# B&R Automation Studio project CControl_Gschneitner (part 2)

### Parameter.typ
```iecst
TYPE
	parAnlage : {REDUND_UNREPLICABLE} 	STRUCT
		Allgemein : {REDUND_UNREPLICABLE} parAllgemein;
		Betrieb : {REDUND_UNREPLICABLE} parBetrieb;
		Ausstattung : {REDUND_UNREPLICABLE} parAusstattung;
		Schrittkette : {REDUND_UNREPLICABLE} parSchrittkette;
		Ventilator1 : {REDUND_UNREPLICABLE} parVentilator;
		Ventilator2 : {REDUND_UNREPLICABLE} parVentilator;
		Boxen : {REDUND_UNREPLICABLE} ARRAY[1..6]OF parBoxen;
		Entfeuchter : {REDUND_UNREPLICABLE} parEntfeuchter;
		Kompressor1 : {REDUND_UNREPLICABLE} parKompressor;
		Kompressor2 : {REDUND_UNREPLICABLE} parKompressor;
		Warmluftofen : {REDUND_UNREPLICABLE} parWarmluftofen;
		Heizregister : {REDUND_UNREPLICABLE} parHeizregister;
		Abluftventilator : {REDUND_UNREPLICABLE} parAbluftventilator;
		Abluftklappe : {REDUND_UNREPLICABLE} parAbluftklappe;
		Umschaltklappen : {REDUND_UNREPLICABLE} parUmschaltklappen;
		Bypassklappe : {REDUND_UNREPLICABLE} parBypassklappe;
		KlappenBoxen : {REDUND_UNREPLICABLE} ARRAY[1..6]OF parKlappenBoxen;
		Notstromaggregat : {REDUND_UNREPLICABLE} parNotstromaggregat;
		Sensoren : {REDUND_UNREPLICABLE} parSensoren;
		Servicebereich : {REDUND_UNREPLICABLE} parServicebereich;
		Fernalarmierung : {REDUND_UNREPLICABLE} parFernalarmierung;
		Scheitholzofen : {REDUND_UNREPLICABLE} parScheitholzofen;
		Tarifabschaltung : {REDUND_UNREPLICABLE} parTarifabschaltung;
		Strombegrenzung : {REDUND_UNREPLICABLE} parStrombegrenzung;
		SchlechtwetterBoxen : {REDUND_UNREPLICABLE} ARRAY[1..6]OF parSchlechtwetterBoxen;
	END_STRUCT;
	parAllgemein : {REDUND_UNREPLICABLE} 	STRUCT
		IPAdresse : {REDUND_UNREPLICABLE} STRING[16];
		SubnetMask : {REDUND_UNREPLICABLE} STRING[16];
		DefaultGateway : {REDUND_UNREPLICABLE} STRING[16];
		HostName : {REDUND_UNREPLICABLE} STRING[16];
		DatumUhrzeitLetzterBetrieb : {REDUND_UNREPLICABLE} DATE_AND_TIME;
		VerzoegerungWarnungen : {REDUND_UNREPLICABLE} REAL;
		VerzoegerungFehler : {REDUND_UNREPLICABLE} REAL;
		StandortHoehe : {REDUND_UNREPLICABLE} REAL;
		AnsaugflaecheVent : {REDUND_UNREPLICABLE} REAL; (*Ansaugfläche des Ventilators (für Luftmengenregelung ohne Entfeuchter)*)
		VerzoegerungAenderungKlappen : {REDUND_UNREPLICABLE} UDINT;
		LoginTimeout : {REDUND_UNREPLICABLE} UDINT;
		VerzUmschBetriebsartBoxen : {REDUND_UNREPLICABLE} UDINT;
		DisplayTimeout : {REDUND_UNREPLICABLE} INT;
		Sprache : {REDUND_UNREPLICABLE} USINT;
		PasswortschutzAus : {REDUND_UNREPLICABLE} BOOL;
		AutoLogoutEin : {REDUND_UNREPLICABLE} BOOL;
		ParameterVorhanden : {REDUND_UNREPLICABLE} BOOL; (*Wenn FALSE, wird beim Neustart der Standardparametersatz geladen*)
	END_STRUCT;
	parBetrieb : {REDUND_UNREPLICABLE} 	STRUCT
		BetriebAutoEin : {REDUND_UNREPLICABLE} BOOL;
	END_STRUCT;
	parAusstattung : {REDUND_UNREPLICABLE} 	STRUCT
		Ventilator1 : {REDUND_UNREPLICABLE} BOOL := TRUE;
		Ventilator2 : {REDUND_UNREPLICABLE} BOOL;
		Entfeuchter : {REDUND_UNREPLICABLE} BOOL;
		EntfeuchterFremd : {REDUND_UNREPLICABLE} BOOL;
		Warmluftofen : {REDUND_UNREPLICABLE} BOOL;
		WarmluftofenBetriebsmldg : {REDUND_UNREPLICABLE} BOOL;
		WarmluftofenTempVorgabe : {REDUND_UNREPLICABLE} BOOL;
		Heizregister : {REDUND_UNREPLICABLE} BOOL;
		HeizregisterDrehzahlvorgabe : {REDUND_UNREPLICABLE} BOOL;
		Scheitholzofen : {REDUND_UNREPLICABLE} BOOL;
		Notstromaggregat : {REDUND_UNREPLICABLE} BOOL;
		Energiemessung : {REDUND_UNREPLICABLE} BOOL;
		Bypassklappe : {REDUND_UNREPLICABLE} BOOL;
		Umschaltklappe1 : {REDUND_UNREPLICABLE} BOOL;
		Umschaltklappe2 : {REDUND_UNREPLICABLE} BOOL;
		Brandschutzklappe : {REDUND_UNREPLICABLE} BOOL;
		Abluftklappe : {REDUND_UNREPLICABLE} BOOL;
		Abluftventilator : {REDUND_UNREPLICABLE} BOOL;
		SensorFrischluft : {REDUND_UNREPLICABLE} BOOL;
		SensorDachluft : {REDUND_UNREPLICABLE} BOOL;
		SensorTrockenluft : {REDUND_UNREPLICABLE} BOOL;
		SensorAbluft : {REDUND_UNREPLICABLE} BOOL;
		SensorLuftgeschwindigkeit : {REDUND_UNREPLICABLE} BOOL;
		SensorKanaldruck : {REDUND_UNREPLICABLE} BOOL;
		Box1 : {REDUND_UNREPLICABLE} BOOL := TRUE;
		Box2 : {REDUND_UNREPLICABLE} BOOL;
		Box3 : {REDUND_UNREPLICABLE} BOOL;
		Box4 : {REDUND_UNREPLICABLE} BOOL;
		Box5 : {REDUND_UNREPLICABLE} BOOL;
		Box6 : {REDUND_UNREPLICABLE} BOOL;
		AlleBoxenklSchliessenWennAus : {REDUND_UNREPLICABLE} BOOL; (*Wenn aktiv, werden alle angesteuerten Boxenklappen im Stillstand geschlossen*)
		MehrereBoxenBelueftbar : {REDUND_UNREPLICABLE} BOOL;
		LuftmngReglerFrischlVent1 : {REDUND_UNREPLICABLE} BOOL; (*Auswahl, ob Luftmengenregelung im Frischluft/Dachluftbetrieb bei Ventilator 1 möglich*)
		LuftmngReglerUmluftVent1 : {REDUND_UNREPLICABLE} BOOL; (*Auswahl, ob Luftmengenregelung im Umluftbetrieb bei Ventilator 1 möglich*)
		LuftmngReglerFrischlVent2 : {REDUND_UNREPLICABLE} BOOL; (*Auswahl, ob Luftmengenregelung im Frischluft/Dachluftbetrieb bei Ventilator 2 möglich*)
		LuftmngReglerUmluftVent2 : {REDUND_UNREPLICABLE} BOOL; (*Auswahl, ob Luftmengenregelung im Umluftbetrieb bei Ventilator 2 möglich*)
		EntfeuchterNurImUmluftbetrieb : {REDUND_UNREPLICABLE} BOOL; (*Betrieb des Entfeuchters ist nur im Umluftbetrieb möglich*)
		BeideVentAusBeiUmschBypasskl : {REDUND_UNREPLICABLE} BOOL; (*Wenn TRUE, wird die Drehzahl beider Ventilatoren bei Umschaltung der Bypassklappe reduziert*)
		BeideVentAusBeiUmschBoxenkl : {REDUND_UNREPLICABLE} BOOL; (*Wenn TRUE, wird die Drehzahl beider Ventilatoren bei Umschaltung der Boxenklappen reduziert*)
		Vent1AusWennUmschUmluftkl : {REDUND_UNREPLICABLE} BOOL; (*Wenn TRUE, wird die Drehzahl von Ventilator 1 bei Umschaltung Umluftklappen reduziert*)
		Vent2AusWennUmschUmluftkl : {REDUND_UNREPLICABLE} BOOL; (*Wenn TRUE, wird die Drehzahl von Ventilator 2 bei Umschaltung Umluftklappen reduziert*)
		AbluftklImFrischlbetrImmerOffen : {REDUND_UNREPLICABLE} BOOL; (*Wenn TRUE, wird die Abluftklappe im Frischluftbetrieb immer geöffnet (im Automatikbetrieb der Klappe)*)
		StellungUmluftklappe1Stillstand : {REDUND_UNREPLICABLE} BOOL; (*FALSE= Frischluft, TRUE= Umluft*)
		StellungUmluftklappe2Stillstand : {REDUND_UNREPLICABLE} BOOL; (*FALSE= Frischluft, TRUE= Umluft*)
		EndlagenVhdUmschaltklappe1 : {REDUND_UNREPLICABLE} BOOL; (*Option Endlagen: Sind keine Endlagen vorhanden, wird die Klappe für die eingestellte Laufzeit umgeschaltet.*)
		EndlagenVhdUmschaltklappe2 : {REDUND_UNREPLICABLE} BOOL; (*Option Endlagen: Sind keine Endlagen vorhanden, wird die Klappe für die eingestellte Laufzeit umgeschaltet.*)
		EndlagenVhdBypassklappe : {REDUND_UNREPLICABLE} BOOL; (*Option Endlagen: Sind keine Endlagen vorhanden, wird die Klappe für die eingestellte Laufzeit umgeschaltet.*)
		EndlagenVhdBoxenklappe1 : {REDUND_UNREPLICABLE} BOOL; (*Option Endlagen: Sind keine Endlagen vorhanden, wird die Klappe für die eingestellte Laufzeit umgeschaltet.*)
		EndlagenVhdBoxenklappe2 : {REDUND_UNREPLICABLE} BOOL; (*Option Endlagen: Sind keine Endlagen vorhanden, wird die Klappe für die eingestellte Laufzeit umgeschaltet.*)
		EndlagenVhdBoxenklappe3 : {REDUND_UNREPLICABLE} BOOL; (*Option Endlagen: Sind keine Endlagen vorhanden, wird die Klappe für die eingestellte Laufzeit umgeschaltet.*)
		EndlagenVhdBoxenklappe4 : {REDUND_UNREPLICABLE} BOOL; (*Option Endlagen: Sind keine Endlagen vorhanden, wird die Klappe für die eingestellte Laufzeit umgeschaltet.*)
		EndlagenVhdBoxenklappe5 : {REDUND_UNREPLICABLE} BOOL; (*Option Endlagen: Sind keine Endlagen vorhanden, wird die Klappe für die eingestellte Laufzeit umgeschaltet.*)
		EndlagenVhdBoxenklappe6 : {REDUND_UNREPLICABLE} BOOL; (*Option Endlagen: Sind keine Endlagen vorhanden, wird die Klappe für die eingestellte Laufzeit umgeschaltet.*)
	END_STRUCT;
	parSchrittkette : {REDUND_UNREPLICABLE} 	STRUCT
		AnlaufverzZweiterVentilator : {REDUND_UNREPLICABLE} UDINT;
		VerzWetterwechsel : {REDUND_UNREPLICABLE} UDINT;
	END_STRUCT;
	parVentilator : {REDUND_UNREPLICABLE} 	STRUCT
		LuftmengeSollFrischluft : {REDUND_UNREPLICABLE} REAL; (*Soll-Luftmenge im Frischluftbetrieb in m³/h pro m² Boxenfläche*)
		LuftmengeSollUmluft : {REDUND_UNREPLICABLE} REAL; (*Soll-Luftmenge im Umluftbetrieb in m³/h pro m² Boxenfläche*)
		LuftmengeBoxMin : {REDUND_UNREPLICABLE} REAL; (*Minimale Lufmenge pro m² Boxenfläche in m³/h*)
		LuftmengeBoxMax : {REDUND_UNREPLICABLE} REAL; (*Maximale Lufmenge pro m² Boxenfläche in m³/h*)
		DrehzahlMin : {REDUND_UNREPLICABLE} REAL; (*Minimale Drehzahl des Ventilators [%]*)
		DrehzahlMax : {REDUND_UNREPLICABLE} REAL; (*Maximale Drehzahl des Ventilators [%]*)
		DrehzahlBeiAuskuehlphase : {REDUND_UNREPLICABLE} REAL; (*Soll-Drehzahl, wenn keine Box aktiv und WLO oder SHO noch in Betrieb [%]*)
		DrzUmschaltung : {REDUND_UNREPLICABLE} REAL; (*Soll-Drehzahl bei Klappenumschaltungen, wenn keine Luftaufbereitung in Betrieb ist [%]*)
		DrzUmschaltungMitLuftaufb : {REDUND_UNREPLICABLE} REAL; (*Soll-Drehzahl bei Klappenumschaltungen, wenn Luftaufbereitung in Betrieb ist [%]*)
		DrehzahlFixUmluft : {REDUND_UNREPLICABLE} REAL; (*Fix-Drehzahl bei Umluftbetrieb [%]*)
		DrehzahlFixFrischluft : {REDUND_UNREPLICABLE} REAL; (*Fix-Drehzahl bei Frischluftbetrieb [%]*)
		DrehzahlStrombegrenzung : {REDUND_UNREPLICABLE} REAL; (*Maximale Drehzahl, wenn Zeitfenster Strombegrenzung aktiv ist [%]*)
		DrehzahlLeistungsreduz : {REDUND_UNREPLICABLE} REAL; (*Maximale Drehzahl, wenn digitaler Eingang für Leistungsreduzierung aktiv ist [%]*)
		P : {REDUND_UNREPLICABLE} REAL;
		I : {REDUND_UNREPLICABLE} REAL;
		D : {REDUND_UNREPLICABLE} REAL;
		D_Filter : {REDUND_UNREPLICABLE} REAL;
		Hysterese : {REDUND_UNREPLICABLE} REAL;
		WindupDaempfung : {REDUND_UNREPLICABLE} REAL;
		Fehlerverzoegerung : {REDUND_UNREPLICABLE} REAL;
		ZeitRampeUp : {REDUND_UNREPLICABLE} UDINT; (*Rampenzeit UP [s]*)
		ZeitRampeDown : {REDUND_UNREPLICABLE} UDINT; (*Rampenzeit DOWN [s]*)
		LuftmengenregUmluftEin : {REDUND_UNREPLICABLE} BOOL; (*Wenn Ein, ist die Luftmengenregelung im Umluftbetrieb aktiv*)
		LuftmengenregFrischluftEin : {REDUND_UNREPLICABLE} BOOL; (*Wenn Ein, ist die Luftmengenregelung im Frischluftbetrieb aktiv*)
	END_STRUCT;
	parBoxen : {REDUND_UNREPLICABLE} 	STRUCT
		StellungKlappe1 : {REDUND_UNREPLICABLE} enumStellungKlappenBoxen; (*0= nicht verwendet, 1= geschlossen, 2= offen*)
		StellungKlappe2 : {REDUND_UNREPLICABLE} enumStellungKlappenBoxen; (*0= nicht verwendet, 1= geschlossen, 2= offen*)
		StellungKlappe3 : {REDUND_UNREPLICABLE} enumStellungKlappenBoxen; (*0= nicht verwendet, 1= geschlossen, 2= offen*)
		StellungKlappe4 : {REDUND_UNREPLICABLE} enumStellungKlappenBoxen; (*0= nicht verwendet, 1= geschlossen, 2= offen*)
		StellungKlappe5 : {REDUND_UNREPLICABLE} enumStellungKlappenBoxen; (*0= nicht verwendet, 1= geschlossen, 2= offen*)
		StellungKlappe6 : {REDUND_UNREPLICABLE} enumStellungKlappenBoxen; (*0= nicht verwendet, 1= geschlossen, 2= offen*)
		Grundflaeche : {REDUND_UNREPLICABLE} REAL; (*Grundfläche Box bei Losetrocknung in m²*)
		NameBox : {REDUND_UNREPLICABLE} STRING[20]; (*Name der Box*)
		Trockengut : {REDUND_UNREPLICABLE} USINT; (*0 = Heu (Lose), 1= Rundballen, 2= Mais, 3= Getreide, 4= Hopfen, 5= Kräuter, 6= Holz*)
		Aus : {REDUND_UNREPLICABLE} BOOL; (*Box Ausgeschaltet*)
		DauerbetriebEin : {REDUND_UNREPLICABLE} BOOL; (*Betriebsart Dauerbetrieb Ein*)
		IntervallbetriebEin : {REDUND_UNREPLICABLE} BOOL; (*Betriebsart Intervallbetrieb Ein*)
		NachtrocknungEin : {REDUND_UNREPLICABLE} BOOL; (*Betriebsart Nachtrocknung Ein*)
		Ventilator1 : {REDUND_UNREPLICABLE} BOOL; (*0= nicht für Box zuständig, 1= für Box zuständig*)
		Ventilator2 : {REDUND_UNREPLICABLE} BOOL; (*0= nicht für Box zuständig, 1= für Box zuständig*)
		Luftentfeuchter : {REDUND_UNREPLICABLE} BOOL; (*0= nicht für Box zuständig, 1= für Box zuständig*)
		Warmluftofen : {REDUND_UNREPLICABLE} BOOL; (*0= nicht für Box zuständig, 1= für Box zuständig*)
		Heizregister : {REDUND_UNREPLICABLE} BOOL; (*0= nicht für Box zuständig, 1= für Box zuständig*)
		Scheitholzofen : {REDUND_UNREPLICABLE} BOOL; (*0= nicht für Box zuständig, 1= für Box zuständig*)
		IntervallbetriebZeiten : {REDUND_UNREPLICABLE} ARRAY[0..23]OF BOOL; (*Zeitbereiche 0-23h Intervallbetrieb*)
		NachtrocknungZeiten : {REDUND_UNREPLICABLE} ARRAY[0..23]OF BOOL; (*Zeitbereiche 0-23h Nachtrocknungsbetrieb*)
	END_STRUCT;
	parZeitfenster : {REDUND_UNREPLICABLE} 	STRUCT
		StartStd : {REDUND_UNREPLICABLE} USINT;
		StartMin : {REDUND_UNREPLICABLE} USINT;
		StoppStd : {REDUND_UNREPLICABLE} USINT;
		StoppMin : {REDUND_UNREPLICABLE} USINT;
	END_STRUCT;
	parEntfeuchter : {REDUND_UNREPLICABLE} 	STRUCT
		Type : {REDUND_UNREPLICABLE} ARRAY[0..14]OF STRING[20];
		Registerflaeche : {REDUND_UNREPLICABLE} ARRAY[0..14]OF REAL;
		EinschaltverzKompressor : {REDUND_UNREPLICABLE} UDINT;
		EinschaltverzAbtau : {REDUND_UNREPLICABLE} UDINT;
		MindestlaufzeitOelsumpf : {REDUND_UNREPLICABLE} UDINT;
		MaxZeitStromlos : {REDUND_UNREPLICABLE} UDINT;
		RestzeitLaufzOelsumpf : {REDUND_UNREPLICABLE} UDINT;
		AnlaufverzModul2 : {REDUND_UNREPLICABLE} UDINT;
		AusschaltverzAbtau : {REDUND_UNREPLICABLE} UDINT;
		LuftgeschwEntfeuchterMin : {REDUND_UNREPLICABLE} REAL; (*Minimale Luftgeschwindigkeit über den Entfeuchter in m/s*)
		LuftgeschwEntfeuchterMax : {REDUND_UNREPLICABLE} REAL; (*Maximale Luftgeschwindigkeit über den Entfeuchter in m/s*)
		EintrittFeuchteEin : {REDUND_UNREPLICABLE} REAL;
		EintrittFeuchteAus : {REDUND_UNREPLICABLE} REAL;
		Dauerbetrieb : {REDUND_UNREPLICABLE} BOOL;
		Automatikbetrieb : {REDUND_UNREPLICABLE} BOOL;
		Aus : {REDUND_UNREPLICABLE} BOOL;
		IndexType : {REDUND_UNREPLICABLE} USINT;
		VerzStandbyHochdruckMax : {REDUND_UNREPLICABLE} UDINT; (*Wenn während Klappenumschaltung oder Strombegrenzung Ventilator Hochdruck überschritten -> Standby*)
		VerzBetriebsmeldung : {REDUND_UNREPLICABLE} UDINT; (*Nur für Fremdgeräte in Verwendung*)
	END_STRUCT;
	parKompressor : {REDUND_UNREPLICABLE} 	STRUCT
		EinschaltverzMagnetventil : {REDUND_UNREPLICABLE} UDINT;
		DrehzahlMin : {REDUND_UNREPLICABLE} REAL;
		DrehzahlMax : {REDUND_UNREPLICABLE} REAL;
		NiederdruckMin : {REDUND_UNREPLICABLE} REAL;
		NiederdruckMax : {REDUND_UNREPLICABLE} REAL;
		RampeDown : {REDUND_UNREPLICABLE} REAL;
		RampeUp : {REDUND_UNREPLICABLE} REAL;
		NiederdruckPumpDown : {REDUND_UNREPLICABLE} REAL;
		DrehzahlFix : {REDUND_UNREPLICABLE} REAL;
		DrehzahlReduzierung : {REDUND_UNREPLICABLE} REAL;
		EintrittTempMin : {REDUND_UNREPLICABLE} REAL;
		EintrittTempMax : {REDUND_UNREPLICABLE} REAL;
		HochdruckMax : {REDUND_UNREPLICABLE} REAL;
		NiederdruckSoll : {REDUND_UNREPLICABLE} REAL;
		Hysterese : {REDUND_UNREPLICABLE} REAL;
		P : {REDUND_UNREPLICABLE} REAL;
		I : {REDUND_UNREPLICABLE} REAL;
		D : {REDUND_UNREPLICABLE} REAL;
		DrehzahlregelungEin : {REDUND_UNREPLICABLE} BOOL;
	END_STRUCT;
	parWarmluftofen : {REDUND_UNREPLICABLE} 	STRUCT
		SaettigungFrischlEin : {REDUND_UNREPLICABLE} REAL;
		WarmlufttempVorgabeSoll : {REDUND_UNREPLICABLE} REAL;
		Hysterese : {REDUND_UNREPLICABLE} REAL;
		Auskuehlzeit : {REDUND_UNREPLICABLE} UDINT;
		VerzBetriebsmeldung : {REDUND_UNREPLICABLE} UDINT;
		VerzWetterwechsel : {REDUND_UNREPLICABLE} UDINT;
		DauerbetriebEin : {REDUND_UNREPLICABLE} BOOL;
		AutomatikbetriebEin : {REDUND_UNREPLICABLE} BOOL;
		Aus : {REDUND_UNREPLICABLE} BOOL;
	END_STRUCT;
	parHeizregister : {REDUND_UNREPLICABLE} 	STRUCT
		VerzWetterwechsel : {REDUND_UNREPLICABLE} UDINT;
		SaettigungFrischlEin : {REDUND_UNREPLICABLE} REAL;
		TrockenluftTempSoll : {REDUND_UNREPLICABLE} REAL;
		Hysterese : {REDUND_UNREPLICABLE} REAL;
		DrehzahlVorgabeMin : {REDUND_UNREPLICABLE} REAL;
		DrehzahlVorgabeMax : {REDUND_UNREPLICABLE} REAL;
		P : {REDUND_UNREPLICABLE} REAL;
		I : {REDUND_UNREPLICABLE} REAL;
		D : {REDUND_UNREPLICABLE} REAL;
		Aus : {REDUND_UNREPLICABLE} BOOL;
		DauerbetriebEin : {REDUND_UNREPLICABLE} BOOL;
		AutomatikbetriebEin : {REDUND_UNREPLICABLE} BOOL;
	END_STRUCT;
	parAbluftventilator : {REDUND_UNREPLICABLE} 	STRUCT
		AbluftfeuchteMax : {REDUND_UNREPLICABLE} REAL;
		Hysterese : {REDUND_UNREPLICABLE} REAL;
		DrehzahlMin : {REDUND_UNREPLICABLE} REAL;
		DrehzahlMax : {REDUND_UNREPLICABLE} REAL;
		P : {REDUND_UNREPLICABLE} REAL;
		I : {REDUND_UNREPLICABLE} REAL;
		D : {REDUND_UNREPLICABLE} REAL;
		Ein : {REDUND_UNREPLICABLE} BOOL;
		Automatik : {REDUND_UNREPLICABLE} BOOL;
	END_STRUCT;
	parAbluftklappe : {REDUND_UNREPLICABLE} 	STRUCT
		Laufzeit : {REDUND_UNREPLICABLE} UDINT;
		AbluftfeuchteMax : {REDUND_UNREPLICABLE} REAL;
		Hysterese : {REDUND_UNREPLICABLE} REAL;
		Automatik : {REDUND_UNREPLICABLE} BOOL;
		Oeffnen : {REDUND_UNREPLICABLE} BOOL;
		Schliessen : {REDUND_UNREPLICABLE} BOOL;
	END_STRUCT;
	parUmschaltklappen : {REDUND_UNREPLICABLE} 	STRUCT
		LaufzeitKlappe1 : {REDUND_UNREPLICABLE} UDINT;
		LaufzeitKlappe2 : {REDUND_UNREPLICABLE} UDINT;
		TemperaturUmschaltung : {REDUND_UNREPLICABLE} REAL;
		Hysterese : {REDUND_UNREPLICABLE} REAL;
		Umschaltverzoegerung : {REDUND_UNREPLICABLE} UDINT;
		TempDifferenzUmschaltung : {REDUND_UNREPLICABLE} REAL;
		Automatik : {REDUND_UNREPLICABLE} BOOL;
		Umluft : {REDUND_UNREPLICABLE} BOOL;
		Frischluft : {REDUND_UNREPLICABLE} BOOL;
	END_STRUCT;
	parBypassklappe : {REDUND_UNREPLICABLE} 	STRUCT
		Laufzeit : {REDUND_UNREPLICABLE} UDINT;
		Automatik : {REDUND_UNREPLICABLE} BOOL;
		Oeffnen : {REDUND_UNREPLICABLE} BOOL;
		Schliessen : {REDUND_UNREPLICABLE} BOOL;
	END_STRUCT;
	parKlappenBoxen : {REDUND_UNREPLICABLE} 	STRUCT
		Laufzeit : {REDUND_UNREPLICABLE} UDINT;
	END_STRUCT;
	parNotstromaggregat : {REDUND_UNREPLICABLE} 	STRUCT
		Vorlaufzeit : {REDUND_UNREPLICABLE} UDINT;
		VerzBetriebsmeldung : {REDUND_UNREPLICABLE} UDINT;
		Nachlaufzeit : {REDUND_UNREPLICABLE} UDINT;
	END_STRUCT;
	parSensoren : {REDUND_UNREPLICABLE} 	STRUCT
		NiederdruckMessberMin : {REDUND_UNREPLICABLE} REAL;
		NiederdruckMessberMax : {REDUND_UNREPLICABLE} REAL;
		HochdruckMessberMin : {REDUND_UNREPLICABLE} REAL;
		HochdruckMessberMax : {REDUND_UNREPLICABLE} REAL;
		EintrittTempMessberMin : {REDUND_UNREPLICABLE} REAL;
		EintrittTempMessberMax : {REDUND_UNREPLICABLE} REAL;
		EintrittFeuchteMessberMin : {REDUND_UNREPLICABLE} REAL;
		EintrittFeuchteMessberMax : {REDUND_UNREPLICABLE} REAL;
		AustrittTempMessberMin : {REDUND_UNREPLICABLE} REAL;
		AustrittTempMessberMax : {REDUND_UNREPLICABLE} REAL;
		AustrittFeuchteMessberMin : {REDUND_UNREPLICABLE} REAL;
		AustrittFeuchteMessberMax : {REDUND_UNREPLICABLE} REAL;
		FrischlTempMessberMin : {REDUND_UNREPLICABLE} REAL;
		FrischlTempMessberMax : {REDUND_UNREPLICABLE} REAL;
		FrischlFeuchteMessberMin : {REDUND_UNREPLICABLE} REAL;
		FrischlFeuchteMessberMax : {REDUND_UNREPLICABLE} REAL;
		DachTempMessberMin : {REDUND_UNREPLICABLE} REAL;
		DachTempMessberMax : {REDUND_UNREPLICABLE} REAL;
		DachFeuchteMessberMin : {REDUND_UNREPLICABLE} REAL;
		DachFeuchteMessberMax : {REDUND_UNREPLICABLE} REAL;
		TrockenlTempMessberMin : {REDUND_UNREPLICABLE} REAL;
		TrockenlTempMessberMax : {REDUND_UNREPLICABLE} REAL;
		TrockenlFeuchteMessberMin : {REDUND_UNREPLICABLE} REAL;
		TrockenlFeuchteMessberMax : {REDUND_UNREPLICABLE} REAL;
		AbluftTempMessberMin : {REDUND_UNREPLICABLE} REAL;
		AbluftTempMessberMax : {REDUND_UNREPLICABLE} REAL;
		AbluftFeuchteMessberMin : {REDUND_UNREPLICABLE} REAL;
		AbluftFeuchteMessberMax : {REDUND_UNREPLICABLE} REAL;
		KanaldruckMessberMin : {REDUND_UNREPLICABLE} REAL;
		KanaldruckMessberMax : {REDUND_UNREPLICABLE} REAL;
		LuftgeschwMessberMin : {REDUND_UNREPLICABLE} REAL;
		LuftgeschwMessberMax : {REDUND_UNREPLICABLE} REAL;
		OffsetNiederdruckModul1 : {REDUND_UNREPLICABLE} REAL;
		OffsetNiederdruckModul2 : {REDUND_UNREPLICABLE} REAL;
		OffsetHochdruckModul1 : {REDUND_UNREPLICABLE} REAL;
		OffsetHochdruckModul2 : {REDUND_UNREPLICABLE} REAL;
		OffsetEintrittTemp : {REDUND_UNREPLICABLE} REAL;
		OffsetEintrittFeuchte : {REDUND_UNREPLICABLE} REAL;
		OffsetAustrittTemp : {REDUND_UNREPLICABLE} REAL;
		OffsetAustrittFeuchte : {REDUND_UNREPLICABLE} REAL;
		OffsetFrischluftTemp : {REDUND_UNREPLICABLE} REAL;
		OffsetFrischluftFeuchte : {REDUND_UNREPLICABLE} REAL;
		OffsetDachTemp : {REDUND_UNREPLICABLE} REAL;
		OffsetDachFeuchte : {REDUND_UNREPLICABLE} REAL;
		OffsetTrockenluftTemp : {REDUND_UNREPLICABLE} REAL;
		OffsetTrockenluftFeuchte : {REDUND_UNREPLICABLE} REAL;
		OffsetAbluftTemp : {REDUND_UNREPLICABLE} REAL;
		OffsetAbluftFeuchte : {REDUND_UNREPLICABLE} REAL;
		OffsetKanaldruck : {REDUND_UNREPLICABLE} REAL;
		OffsetLuftgeschw : {REDUND_UNREPLICABLE} REAL;
		FilterzeitNiederdruck : {REDUND_UNREPLICABLE} UINT;
		FilterzeitHochdruck : {REDUND_UNREPLICABLE} UINT;
		FilterzeitEintritt : {REDUND_UNREPLICABLE} UINT;
		FilterzeitAustritt : {REDUND_UNREPLICABLE} UINT;
		FilterzeitFrischluft : {REDUND_UNREPLICABLE} UINT;
		FilterzeitDachluft : {REDUND_UNREPLICABLE} UINT;
		FilterzeitTrockenluft : {REDUND_UNREPLICABLE} UINT;
		FilterzeitAbluft : {REDUND_UNREPLICABLE} UINT;
		FilterzeitKanaldruck : {REDUND_UNREPLICABLE} UINT;
		FilterzeitLuftgeschwindigkeit : {REDUND_UNREPLICABLE} UINT;
	END_STRUCT;
	parServicebereich : {REDUND_UNREPLICABLE} 	STRUCT
		KontrollintervallUhrzeit : {REDUND_UNREPLICABLE} UDINT;
	END_STRUCT;
	parFernalarmierung : {REDUND_UNREPLICABLE} 	STRUCT
		MailAdresse : {REDUND_UNREPLICABLE} ARRAY[0..3]OF STRING[80];
		EMailAlarmierungEin : {REDUND_UNREPLICABLE} BOOL;
	END_STRUCT;
	parScheitholzofen : {REDUND_UNREPLICABLE} 	STRUCT
		Auskuehlzeit : {REDUND_UNREPLICABLE} UDINT;
	END_STRUCT;
	parTarifabschaltung : {REDUND_UNREPLICABLE} 	STRUCT
		Zeitfenster : {REDUND_UNREPLICABLE} parZeitfenster;
		VorlaufzeitAbschaltungLuftaufb : {REDUND_UNREPLICABLE} USINT;
	END_STRUCT;
	parStrombegrenzung : {REDUND_UNREPLICABLE} 	STRUCT
		Zeitfenster : {REDUND_UNREPLICABLE} parZeitfenster;
	END_STRUCT;
	parSchlechtwetterBoxen : {REDUND_UNREPLICABLE} 	STRUCT
		Stufe : {REDUND_UNREPLICABLE} ARRAY[1..6]OF parSchlechtwetterBoxenStufen;
		HystereseGrenzwert : {REDUND_UNREPLICABLE} REAL;
		AuswahlSensorGrenzwert : {REDUND_UNREPLICABLE} USINT; (*Option Auswahl zuständiger Sensor für Grenzwert (0= Frischluft, 1= Dachluft, 2= Trockenluft)*)
		MaterialfeuchteIst : {REDUND_UNREPLICABLE} USINT; (*Aktuell Materialfeuchte (Trockengutfeuchte) der Box (%)*)
	END_STRUCT;
	parSchlechtwetterBoxenStufen : {REDUND_UNREPLICABLE} 	STRUCT
		Saettigungsdefizit : {REDUND_UNREPLICABLE} REAL; (*Grenzwert Sättigungsdefizit Schlechtwetter [g/m³]*)
		SchlechtwetterZeitLauf : {REDUND_UNREPLICABLE} UDINT; (*Laufzeit bei Schlechtwetter [ms]*)
		SchlechtwetterZeitPause : {REDUND_UNREPLICABLE} UDINT; (*Pausenzeit bei Schlechtwetter [ms]*)
		MaterialfeuchteStufe : {REDUND_UNREPLICABLE} UINT; (*Max. Trockengutfeuchte der Stufe (%)*)
	END_STRUCT;
END_TYPE
```

### Enumeration.typ
```iecst
TYPE
	enumStatusmeldungen :
		(
		STATUSMLDG_STILLSTAND := 0,
		STATUSMLDG_TESTBETRIEB := 1,
		STATUSMLDG_AUTOMATIKBETRIEB := 2,
		STATUSMLDG_DAUERBETRIEB := 3,
		STATUSMLDG_VENTILATOR_EIN := 4,
		STATUSMLDG_VENTILATOR_INTERV := 5
		);
	enumStatus :
		(
		STATUS_NICHT_VERFUEGBAR := 0,
		STATUS_STILLSTAND := 1,
		STATUS_TESTBETRIEB := 2,
		STATUS_DAUERBETRIEB := 3,
		STATUS_INTERVALL_LAUF := 4,
		STATUS_INTERVALL_PAUSE := 5,
		STATUS_NACHTROCKNUNG_LAUF := 6,
		STATUS_NACHTROCKNUNG_PAUSE := 7,
		STATUS_BEREIT := 8,
		STATUS_STOERUNG := 9,
		STATUS_AKTIV := 10,
		STATUS_NICHT_AKTIV := 11,
		STATUS_OFFEN := 12,
		STATUS_GESCHLOSSEN := 13,
		STATUS_NICHT_FREIGEGEBEN := 14,
		STATUS_UNBEKANNT := 15,
		STATUS_IN_BEWEGUNG := 16,
		STATUS_ENTF_ABTAUUNG := 17,
		STATUS_ANLAGE_IN_BETRIEB := 18,
		STATUS_AUSKUEHLPHASE := 19,
		STATUS_ENTF_STANDBY := 20,
		STATUS_KLAPPE_FRISCHLUFT := 21,
		STATUS_KLAPPE_DACHLUFT := 22,
		STATUS_KLAPPE_UMLUFT := 23,
		STATUS_DAUERBETRIEB_PAUSIERT := 24,
		STATUS_SCHLECHTWETTER_LAUF := 25,
		STATUS_SCHLECHTWETTER_PAUSE := 26
		);
	enumBetriebsmodus :
		(
		STILLSTAND := 0,
		BETRIEB := 1,
		IOTEST := 2
		);
	enumWarnung :
		(
		WARNUNG_HOCHDRUCK_MAX_MOD1 := 0,
		WARNUNG_HOCHDRUCK_MAX_MOD2 := 1,
		WARNUNG_SENSOR_AUSTRITT := 2,
		WARNUNG_HEIZREGISTER_FROSTSCHUTZ := 3
		);
	enumFehler :
		(
		FEHLER_24VDC := 0,
		FEHLER_FU_KOMPRESSOR_MODUL1 := 1,
		FEHLER_FU_KOMPRESSOR_MODUL2 := 2,
		FEHLER_BETRIEBSMLDG_KOMPR_MOD1 := 3,
		FEHLER_BETRIEBSMLDG_KOMPR_MOD2 := 4,
		FEHLER_BETRIEBSMLDG_VENTILATOR1 := 5,
		FEHLER_BETRIEBSMLDG_VENTILATOR2 := 6,
		FEHLER_BETRIEBSMLDG_ABLUFTVENT := 7,
		FEHLER_HOCHDRUCK_MODUL1 := 8,
		FEHLER_HOCHDRUCK_MODUL2 := 9,
		FEHLER_NIEDERDRUCK_MODUL1 := 10,
		FEHLER_NIEDERDRUCK_MODUL2 := 11,
		FEHLER_OELDRUCK_KOMPR_MOD1 := 12,
		FEHLER_OELDRUCK_KOMPR_MOD2 := 13,
		FEHLER_KOPFTEMP_KOMPR_MOD1 := 14,
		FEHLER_KOPFTEMP_KOMPR_MOD2 := 15,
		FEHLER_VOLLSCHUTZ_KOMPR_MOD1 := 16,
		FEHLER_VOLLSCHUTZ_KOMPR_MOD2 := 17,
		FEHLER_BETRIEBSMLDG_WARMLUFTOFEN := 18,
		FEHLER_BETRIEBSMLDG_NOTSTROM := 19,
		FEHLER_SENSOR_FRISCHLUFT := 20,
		FEHLER_SENSOR_DACHLUFT := 21,
		FEHLER_SENSOR_TROCKENLUFT := 22,
		FEHLER_SENSOR_ABLUFT := 23,
		FEHLER_SENSOR_EINTRITT := 24,
		FEHLER_SENSOR_AUSTRITT := 25,
		FEHLER_SENSOR_LUFTGESCHW := 26,
		FEHLER_SENSOR_KANALDRUCK := 27,
		FEHLER_SENSOR_NIEDERDRUCK_MOD1 := 28,
		FEHLER_SENSOR_NIEDERDRUCK_MOD2 := 29,
		FEHLER_SENSOR_HOCHDRUCK_MOD1 := 30,
		FEHLER_SENSOR_HOCHDRUCK_MOD2 := 31,
		FEHLER_ENDLAGEN_BYPASSKLAPPE := 32,
		FEHLER_ENDLAGEN_UMSCHALTKLAPPE1 := 33,
		FEHLER_ENDLAGEN_UMSCHALTKLAPPE2 := 34,
		FEHLER_ENDLAGEN_BOXENKLAPPE_1 := 35,
		FEHLER_ENDLAGEN_BOXENKLAPPE_2 := 36,
		FEHLER_ENDLAGEN_BOXENKLAPPE_3 := 37,
		FEHLER_ENDLAGEN_BOXENKLAPPE_4 := 38,
		FEHLER_ENDLAGEN_BOXENKLAPPE_5 := 39,
		FEHLER_ENDLAGEN_BOXENKLAPPE_6 := 40,
		FEHLER_ENDLAGEN_ABLUFTKLAPPE := 41,
		FEHLER_EINTRITT_TEMP_ZU_HOCH := 42,
		FEHLER_EINTRITT_TEMP_ZU_NIEDRIG := 43,
		FEHLER_LZ_PUMPDOWN_MOD1 := 44,
		FEHLER_LZ_PUMPDOWN_MOD2 := 45,
		FEHLER_DREHFELD := 46,
		FEHLER_ENTF_FREMD_STOERMELDUNG := 47,
		FEHLER_ENTF_FREMD_BETRMLDG := 48
		);
	enumAktor :
		(
		AKTOR_SCHRITTKETTE := 0,
		AKTOR_OELSUMPFHEIZUNG_MOD1 := 1,
		AKTOR_OELSUMPFHEIZUNG_MOD2 := 2,
		AKTOR_KOMPRESSOR_MOD1 := 3,
		AKTOR_KOMPRESSOR_MOD2 := 4,
		AKTOR_VENTILATOR_1 := 5,
		AKTOR_VENTILATOR_2 := 6,
		AKTOR_BYPASSKLAPPE := 7,
		AKTOR_UMSCHALTKLAPPE_1 := 8,
		AKTOR_UMSCHALTKLAPPE_2 := 9,
		AKTOR_MAGNETVENTIL_MOD1 := 10,
		AKTOR_MAGNETVENTIL_MOD2 := 11,
		AKTOR_KLAPPE_BOX_1 := 12,
		AKTOR_KLAPPE_BOX_2 := 13,
		AKTOR_KLAPPE_BOX_3 := 14,
		AKTOR_KLAPPE_BOX_4 := 15,
		AKTOR_KLAPPE_BOX_5 := 16,
		AKTOR_KLAPPE_BOX_6 := 17,
		AKTOR_ABLUFTKLAPPE := 18,
		AKTOR_ABLUFTVENTILATOR := 19,
		AKTOR_WARMLUFTOFEN := 20,
		AKTOR_HEIZREGISTER := 21,
		AKTOR_SCHEITHOLZOFEN := 22,
		AKTOR_NOTSTROMAGGREGAT := 23,
		AKTOR_BRANDSCHUTZKLAPPE := 24,
		AKTOR_ENTFEUCHTER_FREMD := 25
		);
	enumSystem :
		(
		FEHLER_IO_TEST_NICHT_FERTIG := 0,
		FEHLER_KOMMUNIKATION_DISPLAY_IO := 1
		);
	enumIcon :
		(
		ICON_VISIBLE := 0,
		ICON_HIDDEN := 1,
		ICON_GRAU := 2,
		ICON_GELB := 3,
		ICON_ROT := 4,
		TEXT_HELLGRAU := 5,
		TEXT_DUNKELGRAU := 6,
		TEXT_GELB := 7,
		TROCKENGUT_HEU_GRAU := 8,
		TROCKENGUT_HEU_GELB := 9,
		TROCKENGUT_RUNDB_GRAU := 10,
		TROCKENGUT_RUNDB_GELB := 11,
		TROCKENGUT_MAIS_GRAU := 12,
		TROCKENGUT_MAIS_GELB := 13,
		TROCKENGUT_GETREIDE_GRAU := 14,
		TROCKENGUT_GETREIDE_GELB := 15,
		TROCKENGUT_HOPFEN_GRAU := 16,
		TROCKENGUT_HOPFEN_GELB := 17,
		TROCKENGUT_KRAEUTER_GRAU := 18,
		TROCKENGUT_KRAEUTER_GELB := 19,
		TROCKENGUT_HOLZ_GRAU := 20,
		TROCKENGUT_HOLZ_GELB := 21,
		TASTE_ENTF_INSELBETR_GESPERRT := 22,
		TASTE_ENTF_INSELBETR_AUS := 23,
		TASTE_ENTF_INSELBETR_EIN := 24
		);
	enumPasswoerter :
		(
		PASSWORT_SPERRE := 0,
		PASSWORT_KUNDE := 4321,
		PASSWORT_LASCO := 21666,
		PASSWORT_ADMIN := 110588,
		PASSWORT_TAN_01 := 222508,
		PASSWORT_TAN_02 := 988036,
		PASSWORT_TAN_03 := 617545,
		PASSWORT_TAN_04 := 548124,
		PASSWORT_TAN_05 := 321642,
		PASSWORT_TAN_06 := 482409,
		PASSWORT_TAN_07 := 679341,
		PASSWORT_TAN_08 := 455576,
		PASSWORT_TAN_09 := 825468,
		PASSWORT_TAN_10 := 959563,
		PASSWORT_TAN_11 := 107316,
		PASSWORT_TAN_12 := 724578,
		PASSWORT_TAN_13 := 804211,
		PASSWORT_TAN_14 := 147228,
		PASSWORT_TAN_15 := 564299,
		PASSWORT_TAN_16 := 832285,
		PASSWORT_TAN_17 := 981185,
		PASSWORT_TAN_18 := 598284,
		PASSWORT_TAN_19 := 730460,
		PASSWORT_TAN_20 := 971962,
		PASSWORT_TAN_21 := 728589,
		PASSWORT_TAN_22 := 396271,
		PASSWORT_TAN_23 := 496146,
		PASSWORT_TAN_24 := 727556,
		PASSWORT_TAN_25 := 110312,
		PASSWORT_TAN_26 := 849433,
		PASSWORT_TAN_27 := 388439,
		PASSWORT_TAN_28 := 907081,
		PASSWORT_TAN_29 := 347765,
		PASSWORT_TAN_30 := 189196,
		PASSWORT_TAN_31 := 129436,
		PASSWORT_TAN_32 := 678825,
		PASSWORT_TAN_33 := 603382,
		PASSWORT_TAN_34 := 752548,
		PASSWORT_TAN_35 := 466127,
		PASSWORT_TAN_36 := 419810,
		PASSWORT_TAN_37 := 628991,
		PASSWORT_TAN_38 := 349832,
		PASSWORT_TAN_39 := 219361,
		PASSWORT_TAN_40 := 257082,
		PASSWORT_TAN_41 := 166753,
		PASSWORT_TAN_42 := 346634,
		PASSWORT_TAN_43 := 635178,
		PASSWORT_TAN_44 := 740794,
		PASSWORT_TAN_45 := 924143,
		PASSWORT_TAN_46 := 162952,
		PASSWORT_TAN_47 := 218710,
		PASSWORT_TAN_48 := 839073,
		PASSWORT_TAN_49 := 423623,
		PASSWORT_TAN_50 := 232733,
		PASSWORT_ZU_GROSS := 999999,
		PASSWORT_ADMIN_1 := 081190,
		PASSWORT_SERVICE := 8613,
		PASSWORT_KUNDE_1 := 1234
		);
	enumPasswortebenen :
		(
		EBENE_SPERRE := 0,
		EBENE_KUNDE := 1,
		EBENE_SERVICE := 2,
		EBENE_LASCO := 3,
		EBENE_ADMIN := 4
		);
	enumSeitenVisu :
		(
		_000_INIT := 0,
		_001_LOGIN := 1,
		_010_HM_UEBERSICHT := 10,
		_100_AL := 100,
		_101_AL := 101,
		_400_IW := 400,
		_401_IW := 401,
		_402_IW := 402,
		_403_IW := 403,
		_404_IW := 404,
		_600_SYS := 600,
		_610_SYS := 610,
		_620_SYS := 620,
		_630_SYS := 630,
		_631_SYS := 631,
		_632_SYS := 632,
		_640_SYS := 640,
		_641_SYS := 641,
		_650_SYS := 650,
		_660_SYS := 660,
		_670_SYS := 670,
		_700_SYS := 700,
		_710_SYS := 710,
		_711_SYS := 711,
		_712_SYS := 712,
		_713_SYS := 713,
		_714_SYS := 714,
		_715_SYS := 715,
		_716_SYS := 716,
		_717_SYS := 717,
		_720_SYS := 720,
		_721_SYS := 721,
		_722_SYS := 722,
		_723_SYS := 723,
		_724_SYS := 724,
		_730_SYS := 730,
		_731_SYS := 731,
		_732_SYS := 732,
		_740_SYS := 740,
		_741_SYS := 741,
		_742_SYS := 742,
		_750_SYS := 750,
		_751_SYS := 751,
		_752_SYS := 752,
		_760_SYS := 760,
		_770_SYS := 770,
		_780_SYS := 780,
		_781_SYS := 781,
		_782_SYS := 782,
		_783_SYS := 783,
		_790_SYS := 790,
		_800_TEST := 800,
		_810_TEST := 810,
		_811_TEST := 811,
		_812_TEST := 812,
		_820_TEST := 820,
		_821_TEST := 821,
		_822_TEST := 822,
		_823_TEST := 823,
		_824_TEST := 824,
		_825_TEST := 825,
		_830_TEST := 830,
		_831_TEST := 831,
		_832_TEST := 832,
		_840_TEST := 840,
		_841_TEST := 841,
		_842_TEST := 842,
		_850_TEST := 850,
		_851_TEST := 851,
		_852_TEST := 852,
		_860_TEST := 860,
		_861_TEST := 861
		);
	enumZusatzmeldungen :
		(
		ZM_STILLSTAND_IOTEST_NICHT_ABGE := 0,
		ZM_STILLSTAND_FEHLER := 1,
		ZM_STILLSTAND_BEREIT := 2,
		ZM_STILLSTAND_ENTF_NOCH_IN_BETR := 3,
		ZM_WARTE_AUF_NOTSTROM := 4,
		ZM_AUSKUEHLZEIT_WLO_AKTIV := 5,
		ZM_AUSKUEHLZEIT_SHO_AKTIV := 6,
		ZM_ANLAUFVERZ_VENT2_AKTIV := 7,
		ZM_ANLAUFVERZ_VENT1_AKTIV := 8,
		ZM_TARIFABSCHALTUNG_AKTIV := 9,
		ZM_STROMBEGRENZUNG_AKTIV := 10,
		ZM_KLAPPEN_WERDEN_UMGESCHALTET := 11,
		ZM_FRISCHLUFTBETRIEB := 12,
		ZM_DACHABSAUGUNGSBETRIEB := 13,
		ZM_UMLUFTBETRIEB := 14,
		ZM_WARTE_AUF_ANFORDERUNG_BOX := 15,
		ZM_STILLSTAND_FEHLERSTOPP := 16,
		ZM_FRISCHLUFTB_VLZ_TARIF := 17,
		ZM_DACHABSAUGUNGSB_VLZ_TARIF := 18,
		ZM_UMLUFTBETR_VLZ_TARIF := 19,
		ZM_INSELBETRIEB_AUS := 20,
		ZM_INSELBETRIEB_STANDBY := 21,
		ZM_INSELBETRIEB_AKTIV := 22,
		ZM_INSELBETRIEB_VENT_NICHT_AKTIV := 23
		);
END_TYPE
```

### VisuIO.typ - Local data types
```iecst
TYPE
	typHmiStatus : {REDUND_UNREPLICABLE} 	STRUCT
		CurUserLevel : {REDUND_UNREPLICABLE} enumPasswortebenen;
		CurPage : {REDUND_UNREPLICABLE} enumSeitenVisu;
		hmiPasswort : {REDUND_UNREPLICABLE} enumPasswoerter;
		Box1 : {REDUND_UNREPLICABLE} typHmiStatusBoxen;
		Box2 : {REDUND_UNREPLICABLE} typHmiStatusBoxen;
		Box3 : {REDUND_UNREPLICABLE} typHmiStatusBoxen;
		Box4 : {REDUND_UNREPLICABLE} typHmiStatusBoxen;
		Box5 : {REDUND_UNREPLICABLE} typHmiStatusBoxen;
		Box6 : {REDUND_UNREPLICABLE} typHmiStatusBoxen;
		Ventilator1 : {REDUND_UNREPLICABLE} typHmiStatusVentilator;
		Ventilator2 : {REDUND_UNREPLICABLE} typHmiStatusVentilator;
		Entfeuchter : {REDUND_UNREPLICABLE} typHmiStatusEntfeuchter;
		WarmluftScheitholzofen : {REDUND_UNREPLICABLE} typHmiStatusWarmluftScheitholz;
		Heizregister : {REDUND_UNREPLICABLE} typHmiStatusHeizregister;
		Brandschutzklappe : {REDUND_UNREPLICABLE} typHmiStatusBrandschutzklappe;
		Umluftklappen : {REDUND_UNREPLICABLE} typHmiStatusUmluftklappen;
		Bypassklappe : {REDUND_UNREPLICABLE} typHmiStatusBypassklappe;
		Abluftklappe : {REDUND_UNREPLICABLE} typHmiStatusAbluftklappe;
		Abluftventilator : {REDUND_UNREPLICABLE} typHmiStatusAbluftventilator;
		Zusatzmeldungen : {REDUND_UNREPLICABLE} typHmiStatusZusatzmeldungen;
		Trendkurven : {REDUND_UNREPLICABLE} typHmiTrendkurven;
		EntfeuchterType : {REDUND_UNREPLICABLE} STRING[20];
		SoftwareVersion : {REDUND_UNREPLICABLE} STRING[16];
		hmiAlarmFilter : {REDUND_UNREPLICABLE} USINT;
		hmiSelectAlarmGroup : {REDUND_UNREPLICABLE} USINT;
		NameSteuerung : {REDUND_UNREPLICABLE} USINT; (*0= LaTronic CControl 4.07, 1= LaTronic CControl 4.07 Plus, 2= LaTronic CControl 3.07, 3= LaTronic CControl 3.04 Plus, 4= HB4000, 5= HB3000,  6= LaTronic CControl 2.07*)
		UserIstAdmin : {REDUND_UNREPLICABLE} BOOL;
		ParameterFileNameAufUsb : {REDUND_UNREPLICABLE} STRING[80];
	END_STRUCT;
	typHmiTrendkurven : {REDUND_UNREPLICABLE} 	STRUCT
		FrischluftTemp : {REDUND_UNREPLICABLE} REAL;
		FrischluftFeuchte : {REDUND_UNREPLICABLE} REAL;
		DachluftTemp : {REDUND_UNREPLICABLE} REAL;
		DachluftFeuchte : {REDUND_UNREPLICABLE} REAL;
		TrockenluftTemp : {REDUND_UNREPLICABLE} REAL;
		TrockenluftFeuchte : {REDUND_UNREPLICABLE} REAL;
		AbluftTemp : {REDUND_UNREPLICABLE} REAL;
		AbluftFeuchte : {REDUND_UNREPLICABLE} REAL;
		EintrittTemp : {REDUND_UNREPLICABLE} REAL;
		EintrittFeuchte : {REDUND_UNREPLICABLE} REAL;
		AustrittTemp : {REDUND_UNREPLICABLE} REAL;
		AustrittFeuchte : {REDUND_UNREPLICABLE} REAL;
		NiederdruckMod1 : {REDUND_UNREPLICABLE} REAL;
		NiederdruckMod2 : {REDUND_UNREPLICABLE} REAL;
		HochdruckMod1 : {REDUND_UNREPLICABLE} REAL;
		HochdruckMod2 : {REDUND_UNREPLICABLE} REAL;
		Luftgeschw : {REDUND_UNREPLICABLE} REAL;
		Kanaldruck : {REDUND_UNREPLICABLE} REAL;
		LeistungAktuell : {REDUND_UNREPLICABLE} REAL;
		CursorTrend1 : {REDUND_UNREPLICABLE} REAL;
		CursorTrend2 : {REDUND_UNREPLICABLE} REAL;
		CursorTrend3 : {REDUND_UNREPLICABLE} REAL;
		WertScrollTrend1 : {REDUND_UNREPLICABLE} REAL;
		WertScrollTrend2 : {REDUND_UNREPLICABLE} REAL;
		WertScrollTrend3 : {REDUND_UNREPLICABLE} REAL;
		WertZoomTrend1 : {REDUND_UNREPLICABLE} REAL;
		WertZoomTrend2 : {REDUND_UNREPLICABLE} REAL;
		WertZoomTrend3 : {REDUND_UNREPLICABLE} REAL;
		ZeitScrollTrend1 : {REDUND_UNREPLICABLE} REAL;
		ZeitScrollTrend2 : {REDUND_UNREPLICABLE} REAL;
		ZeitScrollTrend3 : {REDUND_UNREPLICABLE} REAL;
		ZeitZoomTrend1 : {REDUND_UNREPLICABLE} REAL;
		ZeitZoomTrend2 : {REDUND_UNREPLICABLE} REAL;
		ZeitZoomTrend3 : {REDUND_UNREPLICABLE} REAL;
	END_STRUCT;
	typHmiStatusZusatzmeldungen : {REDUND_UNREPLICABLE} 	STRUCT
		Statustext : {REDUND_UNREPLICABLE} enumZusatzmeldungen;
		RestzeitSchrittAktuell : {REDUND_UNREPLICABLE} UDINT;
		AusgabefeldRestzeit : {REDUND_UNREPLICABLE} enumIcon;
		IconSanduhr : {REDUND_UNREPLICABLE} enumIcon;
	END_STRUCT;
	typHmiStatusBoxen : {REDUND_UNREPLICABLE} 	STRUCT
		Statustext : {REDUND_UNREPLICABLE} enumStatus;
		FarbeStatustext : {REDUND_UNREPLICABLE} enumIcon;
		HintergrundAktiv : {REDUND_UNREPLICABLE} enumIcon;
		HintergrundInaktiv : {REDUND_UNREPLICABLE} enumIcon;
		StatusfeldAktiv : {REDUND_UNREPLICABLE} enumIcon;
		StatusfeldInaktiv : {REDUND_UNREPLICABLE} enumIcon;
		Trockengut : {REDUND_UNREPLICABLE} enumIcon;
		AnzeigeLaufRestzeit : {REDUND_UNREPLICABLE} enumIcon;
		FarbeTextNameBox : {REDUND_UNREPLICABLE} enumIcon;
		TextindexLaufzeit : {REDUND_UNREPLICABLE} USINT;
		LaufRestzeitStunden : {REDUND_UNREPLICABLE} UINT;
		LaufRestzeitMinuten : {REDUND_UNREPLICABLE} UINT;
		IconWitterung : {REDUND_UNREPLICABLE} USINT; (*0= Gute Witterung, 1= Schlechte Witterung*)
	END_STRUCT;
	typHmiStatusVentilator : {REDUND_UNREPLICABLE} 	STRUCT
		TextFrischluftDachluft : {REDUND_UNREPLICABLE} USINT;
		LuftmengenregFrischlSperre : {REDUND_UNREPLICABLE} BOOL;
		LuftmengenregUmluftSperre : {REDUND_UNREPLICABLE} BOOL;
		Status : {REDUND_UNREPLICABLE} enumStatus;
		FarbeIcon : {REDUND_UNREPLICABLE} enumIcon;
		IstDrehzahl : {REDUND_UNREPLICABLE} REAL;
		BargraphInaktiv : {REDUND_UNREPLICABLE} enumIcon;
		BargraphAktiv : {REDUND_UNREPLICABLE} enumIcon;
		FarbeDrehzahl : {REDUND_UNREPLICABLE} enumIcon;
		EingabefeldFixdrehzUmluft : {REDUND_UNREPLICABLE} enumIcon;
		EingabefeldFixdrehzFrischl : {REDUND_UNREPLICABLE} enumIcon;
		EingabefeldLuftmengeUmluft : {REDUND_UNREPLICABLE} enumIcon;
		EingabefeldLuftmengeFrischl : {REDUND_UNREPLICABLE} enumIcon;
		Umluftbetrieb : {REDUND_UNREPLICABLE} enumIcon;
		Luftmenge : {REDUND_UNREPLICABLE} enumIcon;
	END_STRUCT;
	typHmiStatusEntfeuchter : {REDUND_UNREPLICABLE} 	STRUCT
		IstDrehzahlKompressor1 : {REDUND_UNREPLICABLE} REAL;
		IstDrehzahlKompressor2 : {REDUND_UNREPLICABLE} REAL;
		Status : {REDUND_UNREPLICABLE} enumStatus;
		FarbeIcon : {REDUND_UNREPLICABLE} enumIcon;
		EingabeFeuchteEinAusSperre : {REDUND_UNREPLICABLE} BOOL;
		FarbeDrehzahl : {REDUND_UNREPLICABLE} enumIcon;
		FarbeTextStatus : {REDUND_UNREPLICABLE} enumIcon;
		StatusfeldAktiv : {REDUND_UNREPLICABLE} enumIcon;
		StatusfeldInaktiv : {REDUND_UNREPLICABLE} enumIcon;
		IconAbtauung : {REDUND_UNREPLICABLE} enumIcon;
		RestlaufzeitOelsumpfh : {REDUND_UNREPLICABLE} UDINT;
		StatusButtonInselbetrieb : {REDUND_UNREPLICABLE} enumIcon;
		IconAnforderungExtern : {REDUND_UNREPLICABLE} enumIcon;
	END_STRUCT;
	typHmiStatusWarmluftScheitholz : {REDUND_UNREPLICABLE} 	STRUCT
		EingabeSattDefizitSperre : {REDUND_UNREPLICABLE} BOOL;
		TextindexUeberschrift : {REDUND_UNREPLICABLE} USINT;
		StatusWarmluftofen : {REDUND_UNREPLICABLE} enumStatus;
		StatusScheitholzofen : {REDUND_UNREPLICABLE} enumStatus;
		FarbeIcon : {REDUND_UNREPLICABLE} enumIcon;
		StatusfeldShoInaktiv : {REDUND_UNREPLICABLE} enumIcon;
		StatusfeldShoAktiv : {REDUND_UNREPLICABLE} enumIcon;
		StatusfeldWloInaktiv : {REDUND_UNREPLICABLE} enumIcon;
		StatusfeldWloAktiv : {REDUND_UNREPLICABLE} enumIcon;
		FarbeStatustextSho : {REDUND_UNREPLICABLE} enumIcon;
		FarbeStatustextWlo : {REDUND_UNREPLICABLE} enumIcon;
	END_STRUCT;
	typHmiStatusHeizregister : {REDUND_UNREPLICABLE} 	STRUCT
		Status : {REDUND_UNREPLICABLE} enumStatus;
		FarbeIcon : {REDUND_UNREPLICABLE} enumIcon;
		StatusfeldAktiv : {REDUND_UNREPLICABLE} enumIcon;
		StatusfeldInaktiv : {REDUND_UNREPLICABLE} enumIcon;
		FarbeStatustext : {REDUND_UNREPLICABLE} enumIcon;
		EingabeSattDefizitSperre : {REDUND_UNREPLICABLE} BOOL;
		IstDrehzahl : {REDUND_UNREPLICABLE} REAL;
	END_STRUCT;
	typHmiStatusBrandschutzklappe : {REDUND_UNREPLICABLE} 	STRUCT
		FarbeStatustext : {REDUND_UNREPLICABLE} enumIcon;
		Status : {REDUND_UNREPLICABLE} enumStatus;
		StatusfeldInaktiv : {REDUND_UNREPLICABLE} enumIcon;
		StatusfeldAktiv : {REDUND_UNREPLICABLE} enumIcon;
	END_STRUCT;
	typHmiStatusUmluftklappen : {REDUND_UNREPLICABLE} 	STRUCT
		Status : {REDUND_UNREPLICABLE} enumStatus;
		StatusfeldAktiv : {REDUND_UNREPLICABLE} enumIcon;
		StatusfeldInaktiv : {REDUND_UNREPLICABLE} enumIcon;
		FarbeStatustext : {REDUND_UNREPLICABLE} enumIcon;
		EingabefeldTempDifferenz : {REDUND_UNREPLICABLE} enumIcon;
		EingabefeldTempUmschaltung : {REDUND_UNREPLICABLE} enumIcon;
		EingabeTempSchaltpunktSperre : {REDUND_UNREPLICABLE} BOOL;
		EingabeTempDifferenzSperre : {REDUND_UNREPLICABLE} BOOL;
		TextindexButton : {REDUND_UNREPLICABLE} USINT; (*0= Automatik, 1= Frischluft, 2= Dachluft, 3= Umluft*)
		IndexBetriebsart : {REDUND_UNREPLICABLE} USINT; (*0= Automatik, 1= Frischluft, 2= Umluft*)
		TextindexEingabeUmschaltpunkt : {REDUND_UNREPLICABLE} USINT;
	END_STRUCT;
	typHmiStatusBypassklappe : {REDUND_UNREPLICABLE} 	STRUCT
		Status : {REDUND_UNREPLICABLE} enumStatus;
		StatusfeldAktiv : {REDUND_UNREPLICABLE} enumIcon;
		StatusfeldInaktiv : {REDUND_UNREPLICABLE} enumIcon;
		FarbeStatustext : {REDUND_UNREPLICABLE} enumIcon;
		TextindexButton : {REDUND_UNREPLICABLE} USINT; (*0= Automatik, 1= Auf, 2= Zu*)
		IndexBetriebsart : {REDUND_UNREPLICABLE} USINT; (*0= Automatik, 1= Auf, 2= Zu*)
	END_STRUCT;
	typHmiStatusAbluftklappe : {REDUND_UNREPLICABLE} 	STRUCT
		Status : {REDUND_UNREPLICABLE} enumStatus;
		StatusfeldAktiv : {REDUND_UNREPLICABLE} enumIcon;
		StatusfeldInaktiv : {REDUND_UNREPLICABLE} enumIcon;
		FarbeStatustext : {REDUND_UNREPLICABLE} enumIcon;
		EingabeMaxAbluftfeuchteSperre : {REDUND_UNREPLICABLE} BOOL;
		TextindexButton : {REDUND_UNREPLICABLE} USINT; (*0= Automatik, 1= Auf, 2= Zu*)
		IndexBetriebsart : {REDUND_UNREPLICABLE} USINT; (*0= Automatik, 1= Auf, 2= Zu*)
	END_STRUCT;
	typHmiStatusAbluftventilator : {REDUND_UNREPLICABLE} 	STRUCT
		Status : {REDUND_UNREPLICABLE} enumStatus;
		StatusfeldAktiv : {REDUND_UNREPLICABLE} enumIcon;
		StatusfeldInaktiv : {REDUND_UNREPLICABLE} enumIcon;
		FarbeStatustext : {REDUND_UNREPLICABLE} enumIcon;
		EingabeMaxAbluftfeuchteSperre : {REDUND_UNREPLICABLE} BOOL;
		TextindexButton : {REDUND_UNREPLICABLE} USINT;
		IndexBetriebsart : {REDUND_UNREPLICABLE} USINT; (*0= Automatik, 1= Ein, 2= Aus*)
	END_STRUCT;
	typHmiSensoren : {REDUND_UNREPLICABLE} 	STRUCT
		FrischluftTemp : {REDUND_UNREPLICABLE} REAL;
		FrischluftFeuchte : {REDUND_UNREPLICABLE} REAL;
		FrischluftSattDefizit : {REDUND_UNREPLICABLE} REAL;
		DachluftTemp : {REDUND_UNREPLICABLE} REAL;
		DachluftFeuchte : {REDUND_UNREPLICABLE} REAL;
		DachluftSattDefizit : {REDUND_UNREPLICABLE} REAL;
		TrockenluftTemp : {REDUND_UNREPLICABLE} REAL;
		TrockenluftFeuchte : {REDUND_UNREPLICABLE} REAL;
		TrockenluftSattDefizit : {REDUND_UNREPLICABLE} REAL;
		AbluftTemp : {REDUND_UNREPLICABLE} REAL;
		AbluftFeuchte : {REDUND_UNREPLICABLE} REAL;
		AbluftSattDefizit : {REDUND_UNREPLICABLE} REAL;
		EintrittTemp : {REDUND_UNREPLICABLE} REAL;
		EintrittFeuchte : {REDUND_UNREPLICABLE} REAL;
		AustrittTemp : {REDUND_UNREPLICABLE} REAL;
		AustrittFeuchte : {REDUND_UNREPLICABLE} REAL;
		NiederdruckModul1 : {REDUND_UNREPLICABLE} REAL;
		HochdruckModul1 : {REDUND_UNREPLICABLE} REAL;
		NiederdruckModul2 : {REDUND_UNREPLICABLE} REAL;
		HochdruckModul2 : {REDUND_UNREPLICABLE} REAL;
		Luftgeschwindigkeit : {REDUND_UNREPLICABLE} REAL;
		LuftmengeAktuell : {REDUND_UNREPLICABLE} REAL;
		KanaldruckmmH2O : {REDUND_UNREPLICABLE} REAL;
		KanaldruckPa : {REDUND_UNREPLICABLE} REAL;
	END_STRUCT;
	typHmiVisibilityTrend : {REDUND_UNREPLICABLE} 	STRUCT
		FrischluftTemp : {REDUND_UNREPLICABLE} enumIcon;
		FrischluftFeuchte : {REDUND_UNREPLICABLE} enumIcon;
		DachluftTemp : {REDUND_UNREPLICABLE} enumIcon;
		DachluftFeuchte : {REDUND_UNREPLICABLE} enumIcon;
		TrockenluftTemp : {REDUND_UNREPLICABLE} enumIcon;
		TrockenluftFeuchte : {REDUND_UNREPLICABLE} enumIcon;
		AbluftTemp : {REDUND_UNREPLICABLE} enumIcon;
		AbluftFeuchte : {REDUND_UNREPLICABLE} enumIcon;
		Luftgeschw : {REDUND_UNREPLICABLE} enumIcon;
		Kanaldruck : {REDUND_UNREPLICABLE} enumIcon;
		EintrittTemp : {REDUND_UNREPLICABLE} enumIcon;
		EintrittFeuchte : {REDUND_UNREPLICABLE} enumIcon;
		AustrittTemp : {REDUND_UNREPLICABLE} enumIcon;
		AustrittFeuchte : {REDUND_UNREPLICABLE} enumIcon;
		NiederdruckMod1 : {REDUND_UNREPLICABLE} enumIcon;
		NiederdruckMod2 : {REDUND_UNREPLICABLE} enumIcon;
		HochdruckMod1 : {REDUND_UNREPLICABLE} enumIcon;
		HochdruckMod2 : {REDUND_UNREPLICABLE} enumIcon;
	END_STRUCT;
	typHmiVisibility : {REDUND_UNREPLICABLE} 	STRUCT
		Allgemein : {REDUND_UNREPLICABLE} typHmiVisibilityAllgemein;
		Layers : {REDUND_UNREPLICABLE} typHmiVisibilityLayers;
		Buttons : {REDUND_UNREPLICABLE} typHmiVisibilityButtons;
		Trend : {REDUND_UNREPLICABLE} typHmiVisibilityTrend;
	END_STRUCT;
	typHmiVisibilityAllgemein : {REDUND_UNREPLICABLE} 	STRUCT
		Testbetrieb : {REDUND_UNREPLICABLE} enumIcon;
		EbeneService : {REDUND_UNREPLICABLE} enumIcon;
		EbeneLasco : {REDUND_UNREPLICABLE} enumIcon;
		UmschaltverzBetriebsartAktiv : {REDUND_UNREPLICABLE} enumIcon;
		Energiemessung : {REDUND_UNREPLICABLE} enumIcon;
		SymbolRegisterUebersicht : {REDUND_UNREPLICABLE} enumIcon;
		SymbolOfenUebersicht : {REDUND_UNREPLICABLE} enumIcon;
		SymbolEntfeuchterFremdUebersicht : {REDUND_UNREPLICABLE} enumIcon;
		SymbolEntfeuchterUebersicht : {REDUND_UNREPLICABLE} enumIcon;
		Luftgeschwindigkeit : {REDUND_UNREPLICABLE} enumIcon;
		Scheitholzofen : {REDUND_UNREPLICABLE} enumIcon;
		Brandschutzklappe : {REDUND_UNREPLICABLE} enumIcon;
		KompressorModul2 : {REDUND_UNREPLICABLE} enumIcon;
		TemperaturvorgWarmluftofen : {REDUND_UNREPLICABLE} enumIcon;
		Warmluftofen : {REDUND_UNREPLICABLE} enumIcon;
		TemperaturvorgHeizregister : {REDUND_UNREPLICABLE} enumIcon;
		Kanaldruck : {REDUND_UNREPLICABLE} enumIcon;
		Abluftventilator : {REDUND_UNREPLICABLE} enumIcon;
		Abluftklappe : {REDUND_UNREPLICABLE} enumIcon;
		Abluft : {REDUND_UNREPLICABLE} enumIcon;
		Dachluft : {REDUND_UNREPLICABLE} enumIcon;
		Trockenluft : {REDUND_UNREPLICABLE} enumIcon;
		Frischluft : {REDUND_UNREPLICABLE} enumIcon;
		Umschaltklappen : {REDUND_UNREPLICABLE} enumIcon;
		Bypassklappe : {REDUND_UNREPLICABLE} enumIcon;
		LaufzRestOelsumpf : {REDUND_UNREPLICABLE} enumIcon;
		Entfeuchter : {REDUND_UNREPLICABLE} enumIcon;
		Box1 : {REDUND_UNREPLICABLE} enumIcon;
		Box2 : {REDUND_UNREPLICABLE} enumIcon;
		Box3 : {REDUND_UNREPLICABLE} enumIcon;
		Box4 : {REDUND_UNREPLICABLE} enumIcon;
		Box5 : {REDUND_UNREPLICABLE} enumIcon;
		Box6 : {REDUND_UNREPLICABLE} enumIcon;
		Ventilator2 : {REDUND_UNREPLICABLE} enumIcon;
		UmluftbetriebVhd : {REDUND_UNREPLICABLE} enumIcon;
		UebersichtKlappen : {REDUND_UNREPLICABLE} enumIcon;
		UebersichtTrocknungsger : {REDUND_UNREPLICABLE} enumIcon;
		HB4000Hide : {REDUND_UNREPLICABLE} enumIcon; (*Objekte, die nur in der Konfiguration HB4000 sichtbar sind*)
		HB4000 : {REDUND_UNREPLICABLE} enumIcon; (*Objekte, die nur in der Konfiguration HB4000 sichtbar sind*)
		EingabeTrockengutfeuchteBox : {REDUND_UNREPLICABLE} enumIcon;
	END_STRUCT;
	typHmiVisibilityLayers : {REDUND_UNREPLICABLE} 	STRUCT
		ErrorDatum : {REDUND_UNREPLICABLE} enumIcon;
		MdgPwSchutzAus : {REDUND_UNREPLICABLE} enumIcon;
		EbeneFehler : {REDUND_UNREPLICABLE} enumIcon;
		EbeneWarnung : {REDUND_UNREPLICABLE} enumIcon;
		MldgDatumFalsch : {REDUND_UNREPLICABLE} enumIcon;
		MldgKontrolleUhrzeit : {REDUND_UNREPLICABLE} enumIcon;
		MldgStockkontrolle : {REDUND_UNREPLICABLE} enumIcon;
		Zeitfenster : {REDUND_UNREPLICABLE} enumIcon;
		DetailansichtBox : {REDUND_UNREPLICABLE} enumIcon;
		UebersichtEineBox : {REDUND_UNREPLICABLE} enumIcon;
		UebersichtZweiBoxen : {REDUND_UNREPLICABLE} enumIcon;
		UebersichtDreiBoxen : {REDUND_UNREPLICABLE} enumIcon;
		UebersichtVierBoxen : {REDUND_UNREPLICABLE} enumIcon;
		UebersichtFuenfBoxen : {REDUND_UNREPLICABLE} enumIcon;
		UebersichtSechsBoxen : {REDUND_UNREPLICABLE} enumIcon;
		UebersichtEinVentilator : {REDUND_UNREPLICABLE} enumIcon;
		UebersichtZweiVentilatoren : {REDUND_UNREPLICABLE} enumIcon;
		DetailansichtVentilatoren : {REDUND_UNREPLICABLE} enumIcon;
		DetailansichtRegister : {REDUND_UNREPLICABLE} enumIcon;
		DetailansichtOfen : {REDUND_UNREPLICABLE} enumIcon;
		DetailansichtEntfeuchterFremd : {REDUND_UNREPLICABLE} enumIcon;
		DetailansichtEntfeuchter : {REDUND_UNREPLICABLE} enumIcon;
		DetailansichtKlappen : {REDUND_UNREPLICABLE} enumIcon;
		DetailansichtSensoren : {REDUND_UNREPLICABLE} enumIcon;
		Trocknungsbilanz : {REDUND_UNREPLICABLE} enumIcon;
		UebersichtInselbetrieb : {REDUND_UNREPLICABLE} enumIcon;
	END_STRUCT;
	typHmiVisibilityButtons : {REDUND_UNREPLICABLE} 	STRUCT
		IntervallEinstellenBoxAktuell : {REDUND_UNREPLICABLE} enumIcon;
		NachtrocknEinstellenBoxAktuell : {REDUND_UNREPLICABLE} enumIcon;
		IOTestOK : {REDUND_UNREPLICABLE} enumIcon;
		AckTestbetrieb : {REDUND_UNREPLICABLE} enumIcon;
		LogoutButton : {REDUND_UNREPLICABLE} enumIcon;
	END_STRUCT;
	typHmiTrocknungsbilanz : {REDUND_UNREPLICABLE} 	STRUCT
		NameBox : {REDUND_UNREPLICABLE} STRING[20];
		LaufzeitGesamt : {REDUND_UNREPLICABLE} UDINT;
		LaufzeitVentilator : {REDUND_UNREPLICABLE} UDINT;
		LaufzeitLuftaufbereitung : {REDUND_UNREPLICABLE} UDINT;
	END_STRUCT;
	typHmiBoxAktuell : {REDUND_UNREPLICABLE} 	STRUCT
		NameBox : {REDUND_UNREPLICABLE} STRING[20]; (*Name der Box*)
		Trockengut : {REDUND_UNREPLICABLE} enumIcon; (*0 = Losetrocknung, 1= Rundballentrocknung, 2= Mais, 3= Getreide*)
		Aus : {REDUND_UNREPLICABLE} BOOL; (*Box Ausgeschaltet*)
		DauerbetriebEin : {REDUND_UNREPLICABLE} BOOL; (*Betriebsart Dauerbetrieb Ein*)
		IntervallbetriebEin : {REDUND_UNREPLICABLE} BOOL;
		NachtrocknungEin : {REDUND_UNREPLICABLE} BOOL;
		SperreDauerbetrieb : {REDUND_UNREPLICABLE} BOOL;
		SperreIntervallbetrieb : {REDUND_UNREPLICABLE} BOOL;
		Status : {REDUND_UNREPLICABLE} enumStatus;
		ZeitbereicheGesperrt : {REDUND_UNREPLICABLE} ARRAY[0..23]OF BOOL;
		Zeitbereiche : {REDUND_UNREPLICABLE} ARRAY[0..23]OF BOOL;
		RestzeitUmschaltverzBetriebsart : {REDUND_UNREPLICABLE} UDINT;
		AnzeigeLaufRestzeit : {REDUND_UNREPLICABLE} enumIcon;
		TextindexLaufzeit : {REDUND_UNREPLICABLE} USINT;
		LaufRestzeitStunden : {REDUND_UNREPLICABLE} UINT;
		LaufRestzeitMinuten : {REDUND_UNREPLICABLE} UINT;
		IconWitterung : {REDUND_UNREPLICABLE} USINT; (*0= Gute Witterung, 1= Schlechte Witterung*)
		TrockengutfeuchteAktuell : {REDUND_UNREPLICABLE} USINT;
	END_STRUCT;
	typIoTest : {REDUND_UNREPLICABLE} 	STRUCT
		DigitalIn : {REDUND_UNREPLICABLE} typIoTestDigitalIn;
		StatusIn : {REDUND_UNREPLICABLE} typIoTestStatusIn;
		DigitalOut : {REDUND_UNREPLICABLE} typIoTestDigitalOut;
		AnalogIn : {REDUND_UNREPLICABLE} typIoTestAnalogIn;
		AnalogOut : {REDUND_UNREPLICABLE} typIoTestAnalogOut;
	END_STRUCT;
	typIoTestDigitalIn : {REDUND_UNREPLICABLE} 	STRUCT
		diVentilator1InBetrieb : {REDUND_UNREPLICABLE} BOOL;
		di24VDCinternIstOk : {REDUND_UNREPLICABLE} BOOL;
		diBox1Offen : {REDUND_UNREPLICABLE} BOOL;
		diBox1Geschl : {REDUND_UNREPLICABLE} BOOL;
		diBox2Offen : {REDUND_UNREPLICABLE} BOOL;
		diBox2Geschl : {REDUND_UNREPLICABLE} BOOL;
		diVentilator2InBetrieb : {REDUND_UNREPLICABLE} BOOL;
		diDrehzahlbegrVentilator1 : {REDUND_UNREPLICABLE} BOOL;
		diDrehzahlbegrVentilator2 : {REDUND_UNREPLICABLE} BOOL;
		diScheitholzofenInBetrieb : {REDUND_UNREPLICABLE} BOOL;
		diWarmluftofenInBetrieb : {REDUND_UNREPLICABLE} BOOL;
		diBox3Offen : {REDUND_UNREPLICABLE} BOOL;
		diBox3Geschl : {REDUND_UNREPLICABLE} BOOL;
		diBox4Offen : {REDUND_UNREPLICABLE} BOOL;
		diBox4Geschl : {REDUND_UNREPLICABLE} BOOL;
		diBox5Offen : {REDUND_UNREPLICABLE} BOOL;
		diBox5Geschl : {REDUND_UNREPLICABLE} BOOL;
		diBox6Offen : {REDUND_UNREPLICABLE} BOOL;
		diBox6Geschl : {REDUND_UNREPLICABLE} BOOL;
		diAbluftventInBetrieb : {REDUND_UNREPLICABLE} BOOL;
		diAbluftklappeOffen : {REDUND_UNREPLICABLE} BOOL;
		diAbluftklappeGeschl : {REDUND_UNREPLICABLE} BOOL;
		diUmschaltklappe1Offen : {REDUND_UNREPLICABLE} BOOL;
		diUmschaltklappe1Geschl : {REDUND_UNREPLICABLE} BOOL;
		diUmschaltklappe2Offen : {REDUND_UNREPLICABLE} BOOL;
		diUmschaltklappe2Geschl : {REDUND_UNREPLICABLE} BOOL;
		diNotstromaggregatInBetrieb : {REDUND_UNREPLICABLE} BOOL;
		diNiederdruckOkModul1 : {REDUND_UNREPLICABLE} BOOL;
		diNiederdruckOkModul2 : {REDUND_UNREPLICABLE} BOOL;
		diHochdruckOkModul1 : {REDUND_UNREPLICABLE} BOOL;
		diHochdruckOkModul2 : {REDUND_UNREPLICABLE} BOOL;
		diKopftempKompressorModul1 : {REDUND_UNREPLICABLE} BOOL;
		diKopftempKompressorModul2 : {REDUND_UNREPLICABLE} BOOL;
		diOeldruckKompressorModul1 : {REDUND_UNREPLICABLE} BOOL;
		diOeldruckKompressorModul2 : {REDUND_UNREPLICABLE} BOOL;
		diVollschutzKompressorModul1 : {REDUND_UNREPLICABLE} BOOL;
		diVollschutzKompressorModul2 : {REDUND_UNREPLICABLE} BOOL;
		diBetriebsmldgKompressorModul1 : {REDUND_UNREPLICABLE} BOOL;
		diBetriebsmldgKompressorModul2 : {REDUND_UNREPLICABLE} BOOL;
		diLeistungsvorgKompressorExtMod1 : {REDUND_UNREPLICABLE} BOOL;
		diBypassklappeGeschl : {REDUND_UNREPLICABLE} BOOL;
		diBypassklappeOffen : {REDUND_UNREPLICABLE} BOOL;
		diAnfEntfeuchterExtern : {REDUND_UNREPLICABLE} BOOL; (*Nur bei 3.04 in Verwendung*)
		diDrehfeldIstKorrekt : {REDUND_UNREPLICABLE} BOOL; (*Nur bei 3.04 in Verwendung*)
		di230VACIstOk : {REDUND_UNREPLICABLE} BOOL; (*Nur bei HB4000 in Verwendung*)
		diEntfeuchterFremdInBetrieb : {REDUND_UNREPLICABLE} BOOL; (*Nur bei HB4000 in Verwendung*)
		diEntfeuchterFremdStoerung : {REDUND_UNREPLICABLE} BOOL; (*Nur bei HB4000 in Verwendung*)
		diTasteTrocknungPausieren : {REDUND_UNREPLICABLE} BOOL; (*Nur bei HB4000 in Verwendung*)
		diHeizregisterFrostschutz : {REDUND_UNREPLICABLE} BOOL; (*Thermostat Heizregister Forstschutz  EIN*)
	END_STRUCT;
	typIoTestStatusIn : {REDUND_UNREPLICABLE} 	STRUCT
		diStatusNiederdruckMinMod1 : {REDUND_UNREPLICABLE} BOOL;
		diStatusNiederdruckMaxMod1 : {REDUND_UNREPLICABLE} BOOL;
		diStatusHochdruckMinMod1 : {REDUND_UNREPLICABLE} BOOL;
		diStatusHochdruckMaxMod1 : {REDUND_UNREPLICABLE} BOOL;
		diStatusNiederdruckMinMod2 : {REDUND_UNREPLICABLE} BOOL;
		diStatusNiederdruckMaxMod2 : {REDUND_UNREPLICABLE} BOOL;
		diStatusHochdruckMinMod2 : {REDUND_UNREPLICABLE} BOOL;
		diStatusHochdruckMaxMod2 : {REDUND_UNREPLICABLE} BOOL;
		diStatusDifferenzdruckMax : {REDUND_UNREPLICABLE} BOOL;
		diStatusDifferenzdruckMin : {REDUND_UNREPLICABLE} BOOL;
		diStatusLuftgeschwDrahtbruch : {REDUND_UNREPLICABLE} BOOL;
		diStatusLuftgeschwMax : {REDUND_UNREPLICABLE} BOOL;
		diStatusLuftgeschwMin : {REDUND_UNREPLICABLE} BOOL;
		diStatusEintrittTempMin : {REDUND_UNREPLICABLE} BOOL;
		diStatusEintrittTempMax : {REDUND_UNREPLICABLE} BOOL;
		diStatusEintrittFeuchteMin : {REDUND_UNREPLICABLE} BOOL;
		diStatusEintrittFeuchteMax : {REDUND_UNREPLICABLE} BOOL;
		diStatusAustrittTempMin : {REDUND_UNREPLICABLE} BOOL;
		diStatusAustrittTempMax : {REDUND_UNREPLICABLE} BOOL;
		diStatusAustrittFeuchteMin : {REDUND_UNREPLICABLE} BOOL;
		diStatusAustrittFeuchteMax : {REDUND_UNREPLICABLE} BOOL;
		diStatusFrischluftFeuchteMax : {REDUND_UNREPLICABLE} BOOL;
		diStatusFrischluftFeuchteMin : {REDUND_UNREPLICABLE} BOOL;
		diStatusFrischluftTempMax : {REDUND_UNREPLICABLE} BOOL;
		diStatusFrischluftTempMin : {REDUND_UNREPLICABLE} BOOL;
		diStatusTrockenluftFeuchteMax : {REDUND_UNREPLICABLE} BOOL;
		diStatusTrockenluftFeuchteMin : {REDUND_UNREPLICABLE} BOOL;
		diStatusTrockenluftTempMax : {REDUND_UNREPLICABLE} BOOL;
		diStatusTrockenluftTempMin : {REDUND_UNREPLICABLE} BOOL;
		diStatusDachluftFeuchteMax : {REDUND_UNREPLICABLE} BOOL;
		diStatusDachluftFeuchteMin : {REDUND_UNREPLICABLE} BOOL;
		diStatusDachluftTempMax : {REDUND_UNREPLICABLE} BOOL;
		diStatusDachluftTempMin : {REDUND_UNREPLICABLE} BOOL;
		diStatusAbluftTempMax : {REDUND_UNREPLICABLE} BOOL;
		diStatusAbluftTempMin : {REDUND_UNREPLICABLE} BOOL;
		diStatusAbluftFeuchteMax : {REDUND_UNREPLICABLE} BOOL;
		diStatusAbluftFeuchteMin : {REDUND_UNREPLICABLE} BOOL;
	END_STRUCT;
	typIoTestDigitalOut : {REDUND_UNREPLICABLE} 	STRUCT
		doVentilator1Ein : {REDUND_UNREPLICABLE} BOOL;
		doTrocknungInBetrieb : {REDUND_UNREPLICABLE} BOOL;
		doFreigabeBox1 : {REDUND_UNREPLICABLE} BOOL;
		doFreigabeBox2 : {REDUND_UNREPLICABLE} BOOL;
		doTrocknungStoerung : {REDUND_UNREPLICABLE} BOOL;
		doVentilator2Ein : {REDUND_UNREPLICABLE} BOOL;
		doWarmluftofenEin : {REDUND_UNREPLICABLE} BOOL;
		doHeizregisterEin : {REDUND_UNREPLICABLE} BOOL;
		doFreigabeBox3 : {REDUND_UNREPLICABLE} BOOL;
		doFreigabeBox4 : {REDUND_UNREPLICABLE} BOOL;
		doFreigabeBox5 : {REDUND_UNREPLICABLE} BOOL;
		doFreigabeBox6 : {REDUND_UNREPLICABLE} BOOL;
		doBrandschutzklappeAuf : {REDUND_UNREPLICABLE} BOOL;
		doAbluftventilatorEin : {REDUND_UNREPLICABLE} BOOL;
		doAbluftklappeFreigabe : {REDUND_UNREPLICABLE} BOOL;
		doUmluftklappe1Freigabe : {REDUND_UNREPLICABLE} BOOL;
		doUmluftklappe2Freigabe : {REDUND_UNREPLICABLE} BOOL;
		doNotstromaggregatEin : {REDUND_UNREPLICABLE} BOOL;
		doKompressorEinModul1 : {REDUND_UNREPLICABLE} BOOL;
		doKompressorEinModul2 : {REDUND_UNREPLICABLE} BOOL;
		doMagnetventilEinModul1 : {REDUND_UNREPLICABLE} BOOL;
		doMagnetventilEinModul2 : {REDUND_UNREPLICABLE} BOOL;
		doOelsumpfheizungEinModul1 : {REDUND_UNREPLICABLE} BOOL;
		doOelsumpfheizungEinModul2 : {REDUND_UNREPLICABLE} BOOL;
		doBypassklappeOeffnen : {REDUND_UNREPLICABLE} BOOL;
		doBypassklappeSchliessen : {REDUND_UNREPLICABLE} BOOL;
		doUmluftklappe1Oeffnen : {REDUND_UNREPLICABLE} BOOL;
		doUmluftklappe1Schliessen : {REDUND_UNREPLICABLE} BOOL;
		doUmluftklappe2Oeffnen : {REDUND_UNREPLICABLE} BOOL;
		doUmluftklappe2Schliessen : {REDUND_UNREPLICABLE} BOOL;
		doAbluftklappeOeffnen : {REDUND_UNREPLICABLE} BOOL;
		doAbluftklappeSchliessen : {REDUND_UNREPLICABLE} BOOL;
		doEntfFremdFreigabe : {REDUND_UNREPLICABLE} BOOL; (*Nur bei HB4000 in Verwendung*)
		doLuftentfeuchterStrombegrEin : {REDUND_UNREPLICABLE} BOOL; (*Nur bei HB4000 in Verwendung*)
	END_STRUCT;
	typIoTestAnalogIn : {REDUND_UNREPLICABLE} 	STRUCT
		aiFrischluftTemperatur : {REDUND_UNREPLICABLE} REAL;
		aiFrischluftFeuchte : {REDUND_UNREPLICABLE} REAL;
		aiTrockenluftTemperatur : {REDUND_UNREPLICABLE} REAL;
		aiTrockenluftFeuchte : {REDUND_UNREPLICABLE} REAL;
		aiAbluftTemperatur : {REDUND_UNREPLICABLE} REAL;
		aiAbluftFeuchte : {REDUND_UNREPLICABLE} REAL;
		aiDachluftTemperatur : {REDUND_UNREPLICABLE} REAL;
		aiDachluftFeuchte : {REDUND_UNREPLICABLE} REAL;
		aiLuftgeschwindigkeit : {REDUND_UNREPLICABLE} REAL;
		aiDifferenzdruck : {REDUND_UNREPLICABLE} REAL;
		aiNiederdruckModul2 : {REDUND_UNREPLICABLE} REAL;
		aiNiederdruckModul1 : {REDUND_UNREPLICABLE} REAL;
		aiHochdruckModul2 : {REDUND_UNREPLICABLE} REAL;
		aiHochdruckModul1 : {REDUND_UNREPLICABLE} REAL;
		aiEintrittTemperatur : {REDUND_UNREPLICABLE} REAL;
		aiEintrittFeuchte : {REDUND_UNREPLICABLE} REAL;
		aiAustrittTemperatur : {REDUND_UNREPLICABLE} REAL;
		aiAustrittFeuchte : {REDUND_UNREPLICABLE} REAL;
	END_STRUCT;
	typIoTestAnalogOut : {REDUND_UNREPLICABLE} 	STRUCT
		aoDrehzahlvorgVentilator1 : {REDUND_UNREPLICABLE} REAL;
		aoTemperaturvorgWarmluftofen : {REDUND_UNREPLICABLE} REAL;
		aoDrehzahlvorgVentilator2 : {REDUND_UNREPLICABLE} REAL;
		aoLeistungsvorgHeizregister : {REDUND_UNREPLICABLE} REAL;
		aoDrehzahlvorgAbluftventilator : {REDUND_UNREPLICABLE} REAL;
		aoDrehzahlvorgKompressorModul1 : {REDUND_UNREPLICABLE} REAL;
		aoDrehzahlvorgKompressorModul2 : {REDUND_UNREPLICABLE} REAL;
	END_STRUCT;
	typHmiButtonsKlappenBoxen : {REDUND_UNREPLICABLE} 	STRUCT
		Klappe1 : {REDUND_UNREPLICABLE} BOOL;
		Klappe2 : {REDUND_UNREPLICABLE} BOOL;
		Klappe3 : {REDUND_UNREPLICABLE} BOOL;
		Klappe4 : {REDUND_UNREPLICABLE} BOOL;
		Klappe5 : {REDUND_UNREPLICABLE} BOOL;
		Klappe6 : {REDUND_UNREPLICABLE} BOOL;
	END_STRUCT;
	typHmiButtons : {REDUND_UNREPLICABLE} 	STRUCT
		IntervallEinstellenBoxAktuell : {REDUND_UNREPLICABLE} BOOL;
		NachtrocknEinstellenAktuell : {REDUND_UNREPLICABLE} BOOL;
		hideDetailansichtBox : {REDUND_UNREPLICABLE} BOOL;
		hideZeitfenster : {REDUND_UNREPLICABLE} BOOL;
		showBox1 : {REDUND_UNREPLICABLE} BOOL;
		showBox2 : {REDUND_UNREPLICABLE} BOOL;
		showBox3 : {REDUND_UNREPLICABLE} BOOL;
		showBox4 : {REDUND_UNREPLICABLE} BOOL;
		showBox5 : {REDUND_UNREPLICABLE} BOOL;
		showBox6 : {REDUND_UNREPLICABLE} BOOL;
		showVentilatoren : {REDUND_UNREPLICABLE} BOOL;
		showEntfeuchterFremd : {REDUND_UNREPLICABLE} BOOL;
		showEntfeuchter : {REDUND_UNREPLICABLE} BOOL;
		showOfen : {REDUND_UNREPLICABLE} BOOL;
		showHeizregister : {REDUND_UNREPLICABLE} BOOL;
		showKlappen : {REDUND_UNREPLICABLE} BOOL;
		showSensoren : {REDUND_UNREPLICABLE} BOOL;
		QuitFehler : {REDUND_UNREPLICABLE} BOOL;
		TestbetriebEin : {REDUND_UNREPLICABLE} BOOL;
		TestbetriebAbbrechen : {REDUND_UNREPLICABLE} BOOL;
		TestbetriebAbschliessen : {REDUND_UNREPLICABLE} BOOL;
		IpParameterSetzen : {REDUND_UNREPLICABLE} BOOL;
		DatenaufzeichnungAufUsb : {REDUND_UNREPLICABLE} BOOL;
		DatenaufzeichnungLoeschen : {REDUND_UNREPLICABLE} BOOL;
		Logout : {REDUND_UNREPLICABLE} BOOL;
		TouchKalibrieren : {REDUND_UNREPLICABLE} BOOL;
		SicherheitshinweisOk : {REDUND_UNREPLICABLE} BOOL;
		ResetEnergieverbrTag : {REDUND_UNREPLICABLE} BOOL;
		ResetServiceUhrzeit : {REDUND_UNREPLICABLE} BOOL;
		ButtonsKlappeBox1 : {REDUND_UNREPLICABLE} typHmiButtonsKlappenBoxen;
		ButtonsKlappeBox2 : {REDUND_UNREPLICABLE} typHmiButtonsKlappenBoxen;
		ButtonsKlappeBox3 : {REDUND_UNREPLICABLE} typHmiButtonsKlappenBoxen;
		ButtonsKlappeBox4 : {REDUND_UNREPLICABLE} typHmiButtonsKlappenBoxen;
		ButtonsKlappeBox5 : {REDUND_UNREPLICABLE} typHmiButtonsKlappenBoxen;
		ButtonsKlappeBox6 : {REDUND_UNREPLICABLE} typHmiButtonsKlappenBoxen;
		changeWarmluftVent2 : {REDUND_UNREPLICABLE} BOOL; (*Kunde Gschneitner: Button Warmluft/Kaltluft Ventilator 2 (frueher Betriebsart Bypassklappe), TRUE = Warmluft*)
		changeBetrArtAbluftvent : {REDUND_UNREPLICABLE} BOOL;
		changeBetrArtAbluftklappe : {REDUND_UNREPLICABLE} BOOL;
		changeWarmluftVent1 : {REDUND_UNREPLICABLE} BOOL; (*Kunde Gschneitner: Button Warmluft/Kaltluft Ventilator 1 (frueher Betriebsart Umluftklappen), TRUE = Warmluft*)
		ParameterVonUsbLaden : {REDUND_UNREPLICABLE} BOOL;
		ParameterAufUsbKopieren : {REDUND_UNREPLICABLE} BOOL;
		TrocknungsbilanzOk : {REDUND_UNREPLICABLE} BOOL;
		changeTrockengutBox1 : {REDUND_UNREPLICABLE} BOOL;
		changeTrockengutBox2 : {REDUND_UNREPLICABLE} BOOL;
		changeTrockengutBox3 : {REDUND_UNREPLICABLE} BOOL;
		changeTrockengutBox4 : {REDUND_UNREPLICABLE} BOOL;
		changeTrockengutBox5 : {REDUND_UNREPLICABLE} BOOL;
		changeTrockengutBox6 : {REDUND_UNREPLICABLE} BOOL;
	END_STRUCT;
	typHmiActions : {REDUND_UNREPLICABLE} 	STRUCT
		cmdChangePageTo : {REDUND_UNREPLICABLE} enumSeitenVisu;
		cmdInselbetriebEntfeuchterEin : {REDUND_UNREPLICABLE} BOOL;
	END_STRUCT;
	typHmiDatenaufzeichnung : {REDUND_UNREPLICABLE} 	STRUCT
		SaveStepNr : {REDUND_UNREPLICABLE} UINT;
		CopyStepNr : {REDUND_UNREPLICABLE} UINT;
		AnzahlFiles : {REDUND_UNREPLICABLE} UDINT;
		AnzahlEintraegeInFile : {REDUND_UNREPLICABLE} UDINT;
	END_STRUCT;
END_TYPE
```

### Global.typ - Globale Datentypen
```iecst
(*=============================================================================================================================================*)
(*==============================STRUKTUREN NUTZUNGSDATEN ==================================================================================*)

TYPE
	typNutzungsdaten : {REDUND_UNREPLICABLE} 	STRUCT
		Allgemein : {REDUND_UNREPLICABLE} typNutzungAllgemein;
		Bst : {REDUND_UNREPLICABLE} typBetriebsstunden;
		BstGes : {REDUND_UNREPLICABLE} typBetriebsstunden;
		Serviceintervalle : {REDUND_UNREPLICABLE} typServiceintervalle;
		Energiemessung : {REDUND_UNREPLICABLE} typEnergiemessung;
		Trocknungsbilanz : {REDUND_UNREPLICABLE} typNutzungTrocknungsbilanz;
	END_STRUCT;
	typNutzungTrocknungsbilanz : {REDUND_UNREPLICABLE} 	STRUCT
		VentStundenBox1 : {REDUND_UNREPLICABLE} UDINT;
		VentStundenBox2 : {REDUND_UNREPLICABLE} UDINT;
		VentStundenBox3 : {REDUND_UNREPLICABLE} UDINT;
		VentStundenBox4 : {REDUND_UNREPLICABLE} UDINT;
		VentStundenBox5 : {REDUND_UNREPLICABLE} UDINT;
		VentStundenBox6 : {REDUND_UNREPLICABLE} UDINT;
		LuftaufbStundenBox1 : {REDUND_UNREPLICABLE} UDINT;
		LuftaufbStundenBox2 : {REDUND_UNREPLICABLE} UDINT;
		LuftaufbStundenBox3 : {REDUND_UNREPLICABLE} UDINT;
		LuftaufbStundenBox4 : {REDUND_UNREPLICABLE} UDINT;
		LuftaufbStundenBox5 : {REDUND_UNREPLICABLE} UDINT;
		LuftaufbStundenBox6 : {REDUND_UNREPLICABLE} UDINT;
		VentMinutenBox1 : {REDUND_UNREPLICABLE} USINT;
		VentMinutenBox2 : {REDUND_UNREPLICABLE} USINT;
		VentMinutenBox3 : {REDUND_UNREPLICABLE} USINT;
		VentMinutenBox4 : {REDUND_UNREPLICABLE} USINT;
		VentMinutenBox5 : {REDUND_UNREPLICABLE} USINT;
		VentMinutenBox6 : {REDUND_UNREPLICABLE} USINT;
		LuftaufbMinutenBox1 : {REDUND_UNREPLICABLE} USINT;
		LuftaufbMinutenBox2 : {REDUND_UNREPLICABLE} USINT;
		LuftaufbMinutenBox3 : {REDUND_UNREPLICABLE} USINT;
		LuftaufbMinutenBox4 : {REDUND_UNREPLICABLE} USINT;
		LuftaufbMinutenBox5 : {REDUND_UNREPLICABLE} USINT;
		LuftaufbMinutenBox6 : {REDUND_UNREPLICABLE} USINT;
	END_STRUCT;
	typNutzungAllgemein : {REDUND_UNREPLICABLE} 	STRUCT
		LetzterModus : {REDUND_UNREPLICABLE} enumBetriebsmodus;
		DatumLetzterBetrieb : {REDUND_UNREPLICABLE} DATE_AND_TIME;
		IoTestAbgeschlossen : {REDUND_UNREPLICABLE} BOOL;
		SetEthernetOk : {REDUND_UNREPLICABLE} BOOL;
	END_STRUCT;
	typBetriebsstunden : {REDUND_UNREPLICABLE} 	STRUCT
		FrischluftbetrStd : {REDUND_UNREPLICABLE} UDINT;
		UmluftbetrStd : {REDUND_UNREPLICABLE} UDINT;
		Ventilator1Std : {REDUND_UNREPLICABLE} UDINT;
		Ventilator2Std : {REDUND_UNREPLICABLE} UDINT;
		Kompressor1Std : {REDUND_UNREPLICABLE} UDINT;
		Kompressor2Std : {REDUND_UNREPLICABLE} UDINT;
		WarmluftofenStd : {REDUND_UNREPLICABLE} UDINT;
		HeizregisterStd : {REDUND_UNREPLICABLE} UDINT;
		ScheitholzofenStd : {REDUND_UNREPLICABLE} UDINT;
		Abtauung1Std : {REDUND_UNREPLICABLE} UDINT;
		Abtauung2Std : {REDUND_UNREPLICABLE} UDINT;
		OelsumpfheizungStd : {REDUND_UNREPLICABLE} UDINT;
		AbluftventStd : {REDUND_UNREPLICABLE} UDINT;
		Box1Std : {REDUND_UNREPLICABLE} UDINT;
		Box2Std : {REDUND_UNREPLICABLE} UDINT;
		Box3Std : {REDUND_UNREPLICABLE} UDINT;
		Box4Std : {REDUND_UNREPLICABLE} UDINT;
		Box5Std : {REDUND_UNREPLICABLE} UDINT;
		Box6Std : {REDUND_UNREPLICABLE} UDINT;
		FrischluftbetrMin : {REDUND_UNREPLICABLE} USINT;
		UmluftbetrMin : {REDUND_UNREPLICABLE} USINT;
		Ventilator1Min : {REDUND_UNREPLICABLE} USINT;
		Ventilator2Min : {REDUND_UNREPLICABLE} USINT;
		Kompressor1Min : {REDUND_UNREPLICABLE} USINT;
		Kompressor2Min : {REDUND_UNREPLICABLE} USINT;
		WarmluftofenMin : {REDUND_UNREPLICABLE} USINT;
		HeizregisterMin : {REDUND_UNREPLICABLE} USINT;
		ScheitholzofenMin : {REDUND_UNREPLICABLE} USINT;
		Abtauung1Min : {REDUND_UNREPLICABLE} USINT;
		Abtauung2Min : {REDUND_UNREPLICABLE} USINT;
		OelsumpfheizungMin : {REDUND_UNREPLICABLE} USINT;
		AbluftventMin : {REDUND_UNREPLICABLE} USINT;
		Box1Min : {REDUND_UNREPLICABLE} USINT;
		Box2Min : {REDUND_UNREPLICABLE} USINT;
		Box3Min : {REDUND_UNREPLICABLE} USINT;
		Box4Min : {REDUND_UNREPLICABLE} USINT;
		Box5Min : {REDUND_UNREPLICABLE} USINT;
		Box6Min : {REDUND_UNREPLICABLE} USINT;
	END_STRUCT;
	typServiceintervalle : {REDUND_UNREPLICABLE} 	STRUCT
		RestzeitKontrolleUhrzeit : {REDUND_UNREPLICABLE} UDINT;
		KontrolleUhrzeitErforderlich : {REDUND_UNREPLICABLE} BOOL;
	END_STRUCT;
	typEnergiemessung : {REDUND_UNREPLICABLE} 	STRUCT
		LeistungAktuell : {REDUND_UNREPLICABLE} REAL;
		EnergieGesamt : {REDUND_UNREPLICABLE} REAL;
		EnergieTag : {REDUND_UNREPLICABLE} REAL;
	END_STRUCT;
END_TYPE

(*=============================================================================================================================================*)
(*==============================STRUKTUREN ANLAGENKOMMANDOS ==============================================================================*)

TYPE
	cmdAnlage : {REDUND_UNREPLICABLE} 	STRUCT
		Test : {REDUND_UNREPLICABLE} BOOL;
		Auto : {REDUND_UNREPLICABLE} BOOL;
		Leistung : {REDUND_UNREPLICABLE} cmdLeistung;
		StoppExtern : {REDUND_UNREPLICABLE} BOOL;
		StartExtern : {REDUND_UNREPLICABLE} BOOL;
		Start : {REDUND_UNREPLICABLE} BOOL;
		Stop : {REDUND_UNREPLICABLE} BOOL;
		FehlerStopp : {REDUND_UNREPLICABLE} BOOL;
		FehlerModul1 : {REDUND_UNREPLICABLE} BOOL;
		FehlerModul2 : {REDUND_UNREPLICABLE} BOOL;
	END_STRUCT;
	cmdLeistung : {REDUND_UNREPLICABLE} 	STRUCT
		DrehzahlVentilator1 : {REDUND_UNREPLICABLE} REAL;
		DrehzahlVentilator2 : {REDUND_UNREPLICABLE} REAL;
		DrehzahlKompressorModul1 : {REDUND_UNREPLICABLE} REAL;
		DrehzahlKompressorModul2 : {REDUND_UNREPLICABLE} REAL;
		DrehzahlAbluftventilator : {REDUND_UNREPLICABLE} REAL;
		DrehzahlHeizregister : {REDUND_UNREPLICABLE} REAL;
	END_STRUCT;
END_TYPE

(*=============================================================================================================================================*)
(*==============================STRUKTUREN ANLAGENSTATUS ==================================================================================*)

TYPE
	statFehler : {REDUND_UNREPLICABLE} 	STRUCT
		WarnungNr : {REDUND_UNREPLICABLE} USINT;
		FehlerNr : {REDUND_UNREPLICABLE} USINT;
		WarnungText : {REDUND_UNREPLICABLE} STRING[140];
		FehlerText : {REDUND_UNREPLICABLE} STRING[140];
		SummeFehler : {REDUND_UNREPLICABLE} BOOL;
		SummeWarnung : {REDUND_UNREPLICABLE} BOOL;
		SummeSystem : {REDUND_UNREPLICABLE} BOOL;
	END_STRUCT;
	statAnlage : {REDUND_UNREPLICABLE} 	STRUCT
		Betrieb : {REDUND_UNREPLICABLE} BOOL;
		Aktor : {REDUND_UNREPLICABLE} ARRAY[0..39]OF enumStatus;
		Fehler : {REDUND_UNREPLICABLE} statFehler;
		DrehzahlVentilator1 : {REDUND_UNREPLICABLE} REAL;
		DrehzahlVentilator2 : {REDUND_UNREPLICABLE} REAL;
		DrehzahlKompressorModul1 : {REDUND_UNREPLICABLE} REAL;
		DrehzahlKompressorModul2 : {REDUND_UNREPLICABLE} REAL;
		FrischluftTemperatur : {REDUND_UNREPLICABLE} REAL;
		FrischluftFeuchte : {REDUND_UNREPLICABLE} REAL;
		DachluftTemperatur : {REDUND_UNREPLICABLE} REAL;
		DachluftFeuchte : {REDUND_UNREPLICABLE} REAL;
		TrockenluftTemperatur : {REDUND_UNREPLICABLE} REAL;
		TrockenluftFeuchte : {REDUND_UNREPLICABLE} REAL;
		AbluftTemperatur : {REDUND_UNREPLICABLE} REAL;
		AbluftFeuchte : {REDUND_UNREPLICABLE} REAL;
		EintrittTemperatur : {REDUND_UNREPLICABLE} REAL;
		EintrittFeuchte : {REDUND_UNREPLICABLE} REAL;
		AustrittTemperatur : {REDUND_UNREPLICABLE} REAL;
		AustrittFeuchte : {REDUND_UNREPLICABLE} REAL;
		Kanaldruck : {REDUND_UNREPLICABLE} REAL;
		Luftgeschwindigkeit : {REDUND_UNREPLICABLE} REAL;
		NiederdruckModul1 : {REDUND_UNREPLICABLE} REAL;
		NiederdruckModul2 : {REDUND_UNREPLICABLE} REAL;
		HochdruckModul1 : {REDUND_UNREPLICABLE} REAL;
		HochdruckModul2 : {REDUND_UNREPLICABLE} REAL;
		LuftmengeAktuell : {REDUND_UNREPLICABLE} REAL;
		UmluftbetriebAktiv : {REDUND_UNREPLICABLE} BOOL;
		FrischluftbetriebAktiv : {REDUND_UNREPLICABLE} BOOL;
		Warmluft1 : {REDUND_UNREPLICABLE} BOOL; (*Kunde Gschneitner: Umschaltklappe 1 / Ventilator 1 steht auf Warmluft (sonst Kaltluft)*)
		Warmluft2 : {REDUND_UNREPLICABLE} BOOL; (*Kunde Gschneitner: Umschaltklappe 2 / Ventilator 2 steht auf Warmluft (sonst Kaltluft)*)
		WarmluftAnforderung : {REDUND_UNREPLICABLE} BOOL; (*Kunde Gschneitner: mind. ein laufender Ventilator steht auf Warmluft*)
		EnergieverbrTag : {REDUND_UNREPLICABLE} REAL;
		EnergieLeistungAkt : {REDUND_UNREPLICABLE} REAL;
		EnergieverbrGes : {REDUND_UNREPLICABLE} REAL;
		Berechnungen : {REDUND_UNREPLICABLE} statBerechnungen;
		RestlaufzeitenBoxen : {REDUND_UNREPLICABLE} statRestlaufzeitenBoxen;
		WetterIstSchlecht : {REDUND_UNREPLICABLE} BOOL;
	END_STRUCT;
	statRestlaufzeitenBoxen : {REDUND_UNREPLICABLE} 	STRUCT
		Box1Stunden : {REDUND_UNREPLICABLE} UINT;
		Box1Minuten : {REDUND_UNREPLICABLE} UINT;
		Box2Stunden : {REDUND_UNREPLICABLE} UINT;
		Box2Minuten : {REDUND_UNREPLICABLE} UINT;
		Box3Stunden : {REDUND_UNREPLICABLE} UINT;
		Box3Minuten : {REDUND_UNREPLICABLE} UINT;
		Box4Stunden : {REDUND_UNREPLICABLE} UINT;
		Box4Minuten : {REDUND_UNREPLICABLE} UINT;
		Box5Stunden : {REDUND_UNREPLICABLE} UINT;
		Box5Minuten : {REDUND_UNREPLICABLE} UINT;
		Box6Stunden : {REDUND_UNREPLICABLE} UINT;
		Box6Minuten : {REDUND_UNREPLICABLE} UINT;
	END_STRUCT;
	statBerechnungen : {REDUND_UNREPLICABLE} 	STRUCT
		FrischluftSattDefizit : {REDUND_UNREPLICABLE} REAL;
		DachluftSattDefizit : {REDUND_UNREPLICABLE} REAL;
		TrockenluftSattDefizit : {REDUND_UNREPLICABLE} REAL;
		AbluftSattDefizit : {REDUND_UNREPLICABLE} REAL;
		Kanaldruck_mmWs : {REDUND_UNREPLICABLE} REAL;
	END_STRUCT;
END_TYPE

(*=============================================================================================================================================*)
(*==============================STRUKTUREN ANDERE ==========================================================================================*)

TYPE
	typSysteminfo : {REDUND_UNREPLICABLE} 	STRUCT
		BatteriestatusCpu : {REDUND_UNREPLICABLE} USINT;
		TempCpu : {REDUND_UNREPLICABLE} UINT;
		TempEnv : {REDUND_UNREPLICABLE} UINT;
		NodeNumber : {REDUND_UNREPLICABLE} USINT;
		SerialNumber : {REDUND_UNREPLICABLE} UDINT;
		IpAdress : {REDUND_UNREPLICABLE} STRING[20];
		ErrEx : {REDUND_UNREPLICABLE} ARRAY[0..11]OF typErrEx;
		ErrorEx : {REDUND_UNREPLICABLE} BOOL;
		ErrExString : {REDUND_UNREPLICABLE} STRING[30];
		ErrExStringMEM : {REDUND_UNREPLICABLE} STRING[30];
	END_STRUCT;
	typErrEx : {REDUND_UNREPLICABLE} 	STRUCT
		Modul : {REDUND_UNREPLICABLE} ARRAY[0..64]OF BOOL;
	END_STRUCT;
	typEchtzeit : {REDUND_UNREPLICABLE} 	STRUCT
		Jahr : {REDUND_UNREPLICABLE} UINT;
		Monat : {REDUND_UNREPLICABLE} USINT;
		Tag : {REDUND_UNREPLICABLE} USINT;
		WoTag : {REDUND_UNREPLICABLE} USINT;
		Stunde : {REDUND_UNREPLICABLE} USINT;
		Minute : {REDUND_UNREPLICABLE} USINT;
		Sekunde : {REDUND_UNREPLICABLE} USINT;
		Milli : {REDUND_UNREPLICABLE} UINT;
		Mikro : {REDUND_UNREPLICABLE} UINT;
		StdMin : {REDUND_UNREPLICABLE} INT;
	END_STRUCT;
END_TYPE

(*=============================================================================================================================================*)
(*==============================STRUKTUREN AKTOREN =========================================================================================*)

TYPE
	typAktoren : {REDUND_UNREPLICABLE} 	STRUCT
		VentUndKlappen : {REDUND_UNREPLICABLE} fbBoxenVentKlappen;
		Abluftklappe : {REDUND_UNREPLICABLE} fbBoxenAbluftkl;
		Abluftventilator : {REDUND_UNREPLICABLE} fbBoxenAbluftvent;
		OelsumpfheizungModul1 : {REDUND_UNREPLICABLE} fbEntfOelsumpfheiz;
		OelsumpfheizungModul2 : {REDUND_UNREPLICABLE} fbEntfOelsumpfheiz;
		KompressorModul1 : {REDUND_UNREPLICABLE} fbEntfKompressor;
		KompressorModul2 : {REDUND_UNREPLICABLE} fbEntfKompressor;
		Warmluftofen : {REDUND_UNREPLICABLE} fbBoxenWLO;
		Heizregister : {REDUND_UNREPLICABLE} fbBoxenHeizreg;
		Notstromaggregat : {REDUND_UNREPLICABLE} fbBoxenNotstrom;
		Scheitholzofen : {REDUND_UNREPLICABLE} fbBoxenSHO;
		Brandschutzklappe : {REDUND_UNREPLICABLE} fbBoxenKlappenanst;
		EntfeuchterFremd : {REDUND_UNREPLICABLE} fbEntfFremd;
	END_STRUCT;
END_TYPE
```

### Global.var - Globale Variablen
```iecst
VAR
	Boxen : {REDUND_UNREPLICABLE} fbBoxenKonfig; (*Baustein Trocknungsboxen*)
	Aktoren : {REDUND_UNREPLICABLE} typAktoren; (*Funktionsbausteine aller Aktoren (Ventilatoren, Trocknungsgeräte, Klappen, ...)*)
	Tarifabschaltung : {REDUND_UNREPLICABLE} fbTrockTarifabsch; (*Funktionsbaustein Tarifabschaltung*)
	Strombegrenzung : {REDUND_UNREPLICABLE} fbTrockStrombegr; (*Funktionsbaustein Strombegrenzung*)
END_VAR
VAR RETAIN
	Betriebsparameter : {REDUND_UNREPLICABLE} parAnlage; (*Betriebsparametersatz*)
END_VAR
VAR
	CONST_ZEIT_TESTPHASE : {REDUND_UNREPLICABLE} USINT := 3; (*max. Betriebsstunden, in denen der Kompressor am Luftentfeuchter gestartet werden kann, ohne dass die Mindestlaufzeit der Ölsumpfheizung abgelaufen ist (Für Inbetriebnahme Kältetechniker)*)
	gModul2Vorhanden : {REDUND_UNREPLICABLE} BOOL; (*Variable wird gesetzt, wenn eine Luftentfeuchter-Type mit 2 Kompressormodulen ausgewählt wird*)
	gAktModus : {REDUND_UNREPLICABLE} enumBetriebsmodus; (*Aktueller Schrittkettenzustand*)
	gStatusAnlage : {REDUND_UNREPLICABLE} statAnlage; (*Anlagenstatus*)
	gCmdAnlage : {REDUND_UNREPLICABLE} cmdAnlage; (*Anlagenkommandos*)
END_VAR
VAR RETAIN
	Nutzungsdaten : {REDUND_UNREPLICABLE} typNutzungsdaten; (*Struktur Betriebsstunden, Brennstoffleistung, etc...*)
END_VAR
VAR
	Echtzeit : {REDUND_UNREPLICABLE} typEchtzeit; (*Echtzeituhr*)
	Systeminfo : {REDUND_UNREPLICABLE} typSysteminfo; (*Struktur Systeminformationen (Batteriestatus, Hardwaremodule, etc...)*)
	DateTime : {REDUND_UNREPLICABLE} DATE_AND_TIME; (*Aktuelle Systemzeit*)
	VERSION : {REDUND_UNREPLICABLE} STRING[16] := 'V2.1.5'; (*Softwareversion*)
END_VAR
VAR RETAIN
	gMindestlaufzOelsumpfOk : {REDUND_UNREPLICABLE} BOOL; (*Variable wird gesetzt, wenn Mindestlaufzeit der Ölsumpfheiung abgelaufen ist.*)
END_VAR
VAR
	gAktuellesPasswort : {REDUND_UNREPLICABLE} UDINT; (*Aktuelles Passwort in der Visu (Benutzeranmeldung)*)
	gWerksparameterLaden : {REDUND_UNREPLICABLE} BOOL; (*Befehl Werksparametersatz laden*)
	gEnergiemessungModulOk : {REDUND_UNREPLICABLE} BOOL; (*Modulüberwachung Energiemessmodul (wird in den IO-Mappings zur Fehlergenerierung verwendet)*)
END_VAR
```

### VisuIO.var - Local variables
```iecst
VAR
	hmiDatenaufzeichnung : {REDUND_UNREPLICABLE} typHmiDatenaufzeichnung;
	hmiStatus : {REDUND_UNREPLICABLE} typHmiStatus;
END_VAR
VAR RETAIN
	hmiBoxAktuell : {REDUND_UNREPLICABLE} typHmiBoxAktuell;
END_VAR
VAR
	hmiTrocknungsbilanz : {REDUND_UNREPLICABLE} typHmiTrocknungsbilanz;
END_VAR
VAR RETAIN
	hmiActions : {REDUND_UNREPLICABLE} typHmiActions;
END_VAR
VAR
	hmiIoTest : {REDUND_UNREPLICABLE} typIoTest;
	hmiParameter : {REDUND_UNREPLICABLE} parAnlage;
	hmiNutzungsdaten : {REDUND_UNREPLICABLE} typNutzungsdaten;
	hmiSensoren : {REDUND_UNREPLICABLE} typHmiSensoren;
	hmiVisibility : {REDUND_UNREPLICABLE} typHmiVisibility;
	hmiButtons : {REDUND_UNREPLICABLE} typHmiButtons;
END_VAR
```

### Package Logical/Libraries - Globale Bibliotheken

### Library Logical/Libraries/LascoMath (IEC, version 1.00.0) - Funktionsblöcke für diverse Berechnungen

#### LascoMath.var - Exportierte Konstanten
```iecst
(********************************************************************
 * COPYRIGHT -- LASCO Heu- und Forsttechnik GmbH
 ********************************************************************
 * Library: LascoMath
 * Datei: LascoMath.var
 * Autor: Rudolf Lachner
 * Erstellt: 3. März 2014
 ********************************************************************
 * Konstanten der Library LascoMath
 ********************************************************************)
VAR CONSTANT
	CONST_MATH_DRUCK_MEERESHOEHE : REAL := 1013.25;
	CONST_MATH_MAX_VALUE : REAL := 9999999.0;
	CONST_MATH_LUFTDRUCK : REAL := 94520.0;
	CONST_MATH_GASKONSTANTE : REAL := 287.0;
	CONST_MATH_TEMP_NORM : REAL := 21.0;
	CONST_MATH_FAKTOR_DEBIMO : REAL := 0.816;
END_VAR
```

#### LascoMath.fun - Exportierte Funktionen und Funktionsblöcke
```iecst
(********************************************************************
 * COPYRIGHT -- LASCO Heu- und Forsttechnik GmbH
 ********************************************************************
 * Library: LascoMath
 * Datei: LascoMath.fun
 * Autor: Rudolf Lachner
 * Erstellt: 3. März 2014
 ********************************************************************
 * Funktionen und Funktionsblöcke der Library LascoMath
 ********************************************************************)

FUNCTION_BLOCK fbMathLuft (*Berechnungen aus Temperatur, Feuchtigkeit und Meereshöhe (Sättigungsdefizit, Luftdruck, Taupunkttemperatur, etc...)*) (*$GROUP=Anwender*)
	VAR_INPUT
		Freigabe : BOOL; (*Freigabe des Funktionsblocks*)
		LuftTemperatur : REAL; (*Aktuelle Temperatur der Umgebungsluft [°C]*)
		LuftRelFeuchte : REAL; (*relative Feuchtigkeit der Umgebungsluft [%]*)
		MeterUeberAdria : REAL; (*Anlagenstandort Höhe [müA]*)
	END_VAR
	VAR_OUTPUT
		LuftAbsoluteFeuchteSatt : REAL; (*Absolute Feuchtigkeit Satt [g/m³]*)
		LuftAbsoluteFeuchte_g_m3 : REAL; (*Absolute Feuchte [g/m³]*)
		LuftdruckUmgebung : REAL; (*Umgebungsdruck [hPa]*)
		LuftDichte : REAL; (*Luftdichte [kg/m³]*)
		LuftAbsoluteFeuchte_g_kg : REAL; (*Absolute Feuchte [g/kg]*)
		LuftDampfdruckSatt : REAL; (*Sättigungsdampfdruck [mbar]*)
		LuftDampfdruckH2O : REAL; (*Wasserdampfdruck [mbar]*)
		TaupunktTemp : REAL; (*Taupunkttemperatur [°C]*)
		LuftSaettigungsdefizit : REAL; (*Sättigungsdefizit [g/m³]*)
	END_VAR
	VAR
		loc_Taupunkttemp : REAL;
	END_VAR
END_FUNCTION_BLOCK

FUNCTION_BLOCK fbMathTrGutGew (*Berechnungen des Trockengutes (spez. Gewicht, Wasserentzug, Gewicht Start, Gewicht Ende...)*) (*$GROUP=Anwender*)
	VAR_INPUT
		Freigabe : BOOL; (*Freigabe des Funktionsblockes*)
		Anlagentyp : BOOL; (*Boxentrocknung = 0 / Ballentrocknung = 1*)
		Boxenflaeche : REAL; (*Grundfläche Trockenbox [m²]*)
		FuellhoeheTrockengut : REAL; (*Füllhöhe Trockengut [m]*)
		GewichtProBallen : REAL; (*Gewicht pro Heuballen [kg]*)
		AnzahlBallen : REAL; (*Anzahl Ballen [Stk]*)
		FeuchteBeiStart : REAL; (*Trockengut- Feuchte bei Start [%]*)
		FeuchteEnde : REAL; (*Gewünschte Feuchte bei Trocknungsende [%]*)
		Trocknungsgut : USINT; (*Heu = 0, Fichte = 1, Buche = 2, Mais = 3, Weizen = 4*)
		VentilatorInBetrieb : BOOL; (*Ventilator 1 oder 2 in Betrieb*)
		WasserentzugProStunde : REAL; (*Aktueller Wasserentzug pro Stunde [kg/h]*)
		sekTick : BOOL; (*Sekundentakt*)
		KorrekturWertFeuchte : REAL; (*Korrekturwert Trockengutfeuchte von Visu [%]*)
		CmdKorrekturFeuchte : BOOL; (*Befehl Korrektur ausführen*)
		KeinStroemungsfuehler : BOOL; (*Kein Strömungsfühler vorhanden*)
		Automatikbetrieb : BOOL; (*Anlage im Automatikbetrieb*)
		RichtzeitAktStufeTage : UDINT; (*Richtzeit der aktuellen Trockengutstufe [Tage]*)
		stdTick : BOOL; (*Stundentakt*)
		WasserentzugSeitStart : REFERENCE TO REAL; (*Wasserentzug aus Trocknungsgut seit Trocknungsstart [kg]*)
		SpezGewichtUser : REAL;
	END_VAR
	VAR_OUTPUT
		FeuchteAktuell : REAL; (*Aktuelle Trockengutfeuchte [%]*)
		TrockengutGewichtAktuell : REAL; (*Aktuelles Trockengutgewicht [kg]*)
		TrockengutSpezGewicht : REAL; (*Trockengut spez. Gewicht [kg/m³]*)
		TrockengutGewichtStart : REAL; (*Trockengut Gewicht bei Trocknungsstart [kg]*)
		TrockengutGewichtSubstanz : REAL; (*Gewicht Trockengut Substanz (bei 0% Feuchte) [kg]*)
		TrockengutGewichtEnde : REAL; (*Trockengut Gewicht bei Trocknungsende [kg]*)
		TrockengutWasserentzug : REAL; (*Gewicht Wasserentzug von Trocknungsstart bis Ende [kg]*)
		RestgewichtWasser : REAL; (*Restliches Gewicht an Wasser, das noch abzutrocknen ist [kg]*)
	END_VAR
	VAR
		loc_TrockengutGewichtEnde : REAL;
		zzEdge00000 : BOOL;
		zzEdge00001 : BOOL;
		zzEdge00002 : BOOL;
		temp2 : REAL;
		temp1 : REAL;
		loc_cmdKorrekturFeuchte : BOOL;
		zzEdge00003 : BOOL;
		firstInit : BOOL;
		RichtzeitAktStufeStunden : UDINT;
		CmdKorrekturFeuchteRicht : BOOL;
		TeilungFeuchteRicht : REAL;
		KorrekturWertFeuchteRicht : REAL;
		FeuchteBeiStartMEM : REAL;
		zzEdge00004 : BOOL;
	END_VAR
END_FUNCTION_BLOCK

FUNCTION_BLOCK fbMathTrLftMenge
	VAR_INPUT
		DrehzVent1 : REAL; (*Aktuelle Drehzahl Ventilator 1 [%]*)
		DrehzVent2 : REAL; (*Aktuelle Drehzahl Ventilator 2 [%]*)
		Freigabe : BOOL; (*Freigabe des Funktionsblockes*)
		Ventilator1Betrieb : BOOL; (*Ventilator 1 in Betrieb*)
		Ventilator2Betrieb : BOOL; (*Ventilator 2 in Betrieb*)
		DrehzRegelungAktiv : BOOL; (*Mengen- oder Druckregelung aktiv*)
		Ventilator12FixDrehzahl : BOOL; (*Ventilator 1 + 2 mit Fixdrehzahl*)
		Ventilator2Manuell : BOOL; (*Ventilator 2 Manuell*)
		Luftgeschw : REAL; (*Aktuelle Luftgeschwindigkeit [m/s]*)
		LuftkanalQuerschnitt : REAL; (*Querschnitt Luftkanal [m²]*)
		ZuluftSattDefizit : REAL; (*Sättigungsdefizit der Zuluft [g/m³]*)
		OffsetWasserentzug : REAL; (*Offset für Wasserentzug pro Stunde*)
		ZweiBoxenSystem : BOOL;
	END_VAR
	VAR_OUTPUT
		LuftmengeAktuell : REAL; (*Aktuelle Luftmenge [m³/h]*)
		WasserentzugProStunde : REAL; (*Wasserentzug pro Stunde [kg/h]*)
	END_VAR
	VAR
		loc_DrehzVerhaeltnis : REAL;
	END_VAR
END_FUNCTION_BLOCK

FUNCTION_BLOCK fbMathTrLftDruck (*Berechnungen mit Drucksensor*) (*$GROUP=Anwender*)
	VAR_INPUT
		Freigabe : BOOL; (*Freigabe des Funktionsblockes*)
		TrockenluftDruck : REAL; (*Überdruck der Trockenluft [Pa]*)
	END_VAR
	VAR_OUTPUT
		LuftDruck_mmWS : REAL; (*Aktueller Luftdruck [mmWS]*)
		LuftDruck_mbar : REAL; (*Aktueller Luftdruck [mbar]*)
		LuftDruck_bar : REAL; (*Aktueller Luftdruck [bar]*)
	END_VAR
END_FUNCTION_BLOCK

FUNCTION_BLOCK fbMathWetter (*Auswertung des aktuellen Wetters anhand Rezept und Sättigungsdefizit*) (*$GROUP=Anwender*)
	VAR_INPUT
		Freigabe : BOOL; (*Freigabe des Funktionsblocks*)
		SattDefizitRezept : REAL; (*Aktuelles Sättigungsdefizit im Rezept [g/m³]*)
		SattDefizitAktuell : REAL; (*Aktuelles Sättigungsdefizit der Frischluft [g/m³]*)
		HystereseUmschaltung : REAL; (*Hysterese für die Wetterumschaltung [g/m³]*)
		ZeitVerzUmschaltung : UDINT; (*Zeitverzögerung Wetterumschaltung [ms]*)
	END_VAR
	VAR_OUTPUT
		WetterGut : BOOL; (*Ausgang Wetter Gut*)
		WetterMittel : BOOL; (*Ausgang Wetter Mittel*)
		WetterSchlecht : BOOL; (*Ausgang Wetter Schlecht*)
	END_VAR
	VAR
		loc_WetterGut : BOOL;
		loc_WetterSchlecht : BOOL;
		TOF_WetterGut : TOF;
		TON_WetterSchlecht : TON;
		TON_WetterGut : TON;
	END_VAR
END_FUNCTION_BLOCK

FUNCTION_BLOCK fbMathMessblende (*Berechnungen für Messkanäle mit Messblende*) (*$GROUP=Anwender*)
	VAR_INPUT
		Enable : BOOL;
		TemperaturAktuell : REAL; (*Aktuelle Temperatur an der Messblende [°C]*)
	END_VAR
	VAR_OUTPUT
		LuftdichteAktuell : REAL;
	END_VAR
	VAR_INPUT
		DifferenzdruckMessblende : REAL; (*[Pa]*)
	END_VAR
	VAR_OUTPUT
		LuftgeschwindigkeitAktuell : REAL; (*[m/s]*)
	END_VAR
	VAR_INPUT
		Kanalquerschnitt : REAL; (*[m²]*)
	END_VAR
	VAR_OUTPUT
		VolumenstromAktuell : REAL; (*[m³/h]*)
		LuftdichteNorm : REAL;
		LuftgeschwindigkeitNorm : REAL;
		VolumenstromNorm : REAL;
	END_VAR
	VAR_INPUT
		LuftgeschwindigkeitSensor : REAL;
	END_VAR
	VAR_OUTPUT
		VolumenstromVergleich : REAL;
	END_VAR
END_FUNCTION_BLOCK
```

#### fbMathLuft.st - Berechnungen aus Temperatur, Feuchtigkeit und Meereshöhe (Sättigungsdefizit, Luftdruck, Taupunkttemperatur, etc...)
```iecst
(********************************************************************
 * COPYRIGHT -- LASCO Heu- und Forsttechnik GmbH
 ********************************************************************
 * Library: LascoMath
 * Datei: fbMathLuft.st
 * Autor: Rudolf Lachner
 * Erstellt: 3. März 2014
 ********************************************************************
 * Implementierung der Library LascoMath
 ********************************************************************)

(* Berechnungen aus Temperatur, Feuchtigkeit und Meereshöhe (Sättigungsdefizit, Luftdruck, Taupunkttemperatur, etc...) *)
FUNCTION_BLOCK fbMathLuft

	IF (Freigabe = TRUE) THEN

		//Luftdruck [hPa]
		LuftdruckUmgebung	:= CONST_MATH_DRUCK_MEERESHOEHE * EXPT(1 - 0.0065 * MeterUeberAdria / 288.15, 5.255);

		//Luftdichte [kg/m³]
		IF (LuftTemperatur <> -273.15) THEN
			LuftDichte	:= (LuftdruckUmgebung * 100) / (287.058 * (273.15 + LuftTemperatur));
		ELSE
			LuftDichte	:= CONST_MATH_MAX_VALUE;
		END_IF

		//Umgebungsluft absolute Feuchte gesättigt [g/m³]
		IF (LuftTemperatur <> -237.3) AND (LuftTemperatur <> -273.15) THEN
			LuftAbsoluteFeuchteSatt		:= 216.67 * ((6.1078 * EXPT(10 , (7.5 * LuftTemperatur / (237.3 + LuftTemperatur)))) / (LuftTemperatur + 273.15));
		ELSE
			LuftAbsoluteFeuchteSatt		:= CONST_MATH_MAX_VALUE;
		END_IF

		//Umgebungsluft absolute Feuchte [g/m³]
		IF (LuftAbsoluteFeuchteSatt < CONST_MATH_MAX_VALUE) THEN
			LuftAbsoluteFeuchte_g_m3	:= (LuftRelFeuchte / 100) * LuftAbsoluteFeuchteSatt;
		ELSE
			LuftAbsoluteFeuchte_g_m3 	:= CONST_MATH_MAX_VALUE;
		END_IF

		//Umgebungsluft Sättigungsdefizit [g/m³]
		IF (LuftAbsoluteFeuchte_g_m3 < CONST_MATH_MAX_VALUE) THEN
			LuftSaettigungsdefizit		:= LuftAbsoluteFeuchteSatt - LuftAbsoluteFeuchte_g_m3;
		ELSE
			LuftSaettigungsdefizit		:= CONST_MATH_MAX_VALUE;
		END_IF

		//Umgebungsluft absolute Feuchte [g/kg]
		IF (LuftAbsoluteFeuchte_g_m3 < CONST_MATH_MAX_VALUE) AND (LuftDichte < CONST_MATH_MAX_VALUE) AND (LuftDichte <> 0) THEN
			LuftAbsoluteFeuchte_g_kg	:= LuftAbsoluteFeuchte_g_m3 / LuftDichte;
		ELSE
			LuftAbsoluteFeuchte_g_kg	:= CONST_MATH_MAX_VALUE;
		END_IF

		//Umgebungsluft Sättigungsdampfdruck [mbar]
		IF (LuftTemperatur <> 237.3) THEN
			LuftDampfdruckSatt		:= 6.09 * EXPT(10, ((7.5 * LuftTemperatur) / (237.3 + LuftTemperatur)));
		ELSE
			LuftDampfdruckSatt		:= CONST_MATH_MAX_VALUE;
		END_IF

		//Umgebungsluft Wasserdampfdruck [mbar]
		IF (LuftDampfdruckSatt < CONST_MATH_MAX_VALUE) THEN
			LuftDampfdruckH2O		:= LuftDampfdruckSatt * (LuftRelFeuchte / 100);
		ELSE
			LuftDampfdruckH2O		:= CONST_MATH_MAX_VALUE;
		END_IF

		//Umgebungsluft Taupunkttemperatur [°C]
		IF (LuftDampfdruckH2O < CONST_MATH_MAX_VALUE) AND (LuftDampfdruckH2O <> 0) THEN
			loc_Taupunkttemp	:= LOG(LuftDampfdruckH2O);
			IF (loc_Taupunkttemp <> 8.233) THEN
				TaupunktTemp	:= (234.67 * loc_Taupunkttemp - 184.2) / (8.233 - loc_Taupunkttemp);
			ELSE
				TaupunktTemp	:= CONST_MATH_MAX_VALUE;
			END_IF
		ELSE
			TaupunktTemp		:= CONST_MATH_MAX_VALUE;
		END_IF

	ELSE

		LuftdruckUmgebung			:= CONST_MATH_MAX_VALUE;
		LuftAbsoluteFeuchteSatt		:= CONST_MATH_MAX_VALUE;
		LuftAbsoluteFeuchte_g_kg	:= CONST_MATH_MAX_VALUE;
		LuftAbsoluteFeuchte_g_m3	:= CONST_MATH_MAX_VALUE;
		LuftDichte					:= CONST_MATH_MAX_VALUE;
		TaupunktTemp				:= CONST_MATH_MAX_VALUE;
		LuftDampfdruckH2O			:= CONST_MATH_MAX_VALUE;
		LuftDampfdruckSatt			:= CONST_MATH_MAX_VALUE;
		LuftSaettigungsdefizit		:= CONST_MATH_MAX_VALUE;

	END_IF

END_FUNCTION_BLOCK
```
